KUKA KRL program: vw_prc_usr_r.src, vw_prc_usr_r.dat

--- vw_prc_usr_r.src ---
&ACCESS RV1
&COMMENT KS26
&REL 200
&PARAM DISKPATH = VW_User/Applikation/LM_Vision/Perceptron
&PARAM TPUSER_VERSION = 8.3.0
DEF vw_prc_usr_r( )
;
;*---------------------------------------------*
;* Perceptron GmbH                             *
;* Version 1.2.0  / VKRC 2 / VKRC 4            *
;*                                             *
;* Bearbeitet am:                              *
;* 21.12.2010 MG                               *
;*     ueberarbeitet auf Stand V1.0.0 / VKRC 4 *
;*                                             *
;* 26.12.2013 HF                               *
;*     512 Kompensations-UP holen neu          *
;*     521 Messpunkte abgeschlossen neu        *
;*     531 Messende mit SPS entfernt           *
;*     512 ist jetzt 514                       *
;*     FLAG-Modell-Kontrolle                   *
;*                                             *
;* 05.02.2014 MG                               *
;*     V1.1.6: VKRC4 mit                       *
;*             Robotertausch                   *
;*             Sensortausch                    *
;*             Compmodell                      *
;*     V1.1.7: Tempcompsystem                  *
;*                                             *
;* 15.07.2015 RB                               *
;*     V1.1.8: Modell-Erweiterung              *
;*             Modell-Flags angepasst          *
;*             UP-Nr.-Zuweiung angepasst       *
;*             Roboter Korrekturframe holen    *
;*                                             *
;* 12.12.2015 DB                               *
;*     Conveyor implementiert                  *
;*                                             *
;* 09.05.2017 HF                               *
;*     PRCP/Init implementiert                 *
;*                                             *
;*     V1.2.0: 524 - Achswinkel speichern      *
;*             525 - Start Messpunkt ID        *
;*                    Sendet Pose-ID           *
;*             SysInit-1  System Init          *
;*             SysInit-2  System Init          *
;*             ModelInit  Modellfreigaben      *
;*             FrameInit Max  VF-Limits        *
;*             FrameInit Min  VF-Limits        *
;*                                             *
;* 01.02.2019 HF                               *
;*     V1.3.0: TPUSER_VERSION = 8.3.0          *
;*                                             *
;*---------------------------------------------*
;
END
;
;FOLD Perceptron Interface
GLOBAL DEF PRC_Interface(USER_CMD:IN,CMD_SEL:IN,FUNKTION:IN,nPAR2:IN,nPAR3:IN,nPAR4:IN,nPAR5:IN,nPAR6:IN,nPAR7:IN,nPAR8:IN,nPAR9:IN)
DECL VW_USER_CMD USER_CMD
DECL INT         CMD_SEL      ; Modus
DECL INT         FUNKTION     ; Funktion
DECL INT         nPAR2
DECL INT         nPAR3
DECL INT         nPAR4
DECL INT         nPAR5
DECL INT         nPAR6
DECL INT         nPAR7
DECL INT         nPAR8
DECL INT         nPAR9
DECL INT         nFlagCounter
DECL INT         I ;allgemeiner Zaehler
DECL KRLMSG_T      USER_MSG
  IF USER_CMD == #USR_MAKRO THEN
     SWITCH CMD_SEL
        CASE 1001 ; PRC_SYSINIT_1      Hauptgruppe 9, Untergruppe 1
           ; System Einstellungen 1
           PRC_SysInit1(FUNKTION,nPAR2,nPAR3,nPAR4,nPAR5,nPAR6)
		     ; Subsystem              Toolkalibrier-Modus = 0-ToolFinder/1=Temperaturkalibrierung
	         ; Conveyortech           0=Ohne/1=Mit
             ; Alive-Bit              0=Ohne/1=Mit
             ; KorrekturBase          (Default 31, Conveyor 11)
		     ; Robotertausch-VF
           ; Frei
        CASE 1002 ; PRC_SYSINIT_2      Hauptgruppe 9, Untergruppe 2
           ; System Einstellungen 2
           PRC_SysInit2(FUNKTION,nPAR2,nPAR3,nPAR4,nPAR5,nPAR6)
		     ; Timeout Messpunkt      [ms]
		     ; Timeout Kommunikation  [ms]
		     ; Start Fehler-Flags
		     ; Start Master-Signale
		     ; Interrupt fuer RobMove
           ; Interrupt fuer RobNoMove
        CASE 1003 ; PRC_MODELINIT      Hauptgruppe 9, Untergruppe 3
           ; Modell Freigaben
           PRC_ModelInit(FUNKTION,nPAR2,nPAR3,nPAR4,nPAR5,nPAR6)
             ; Freigegebenes Modell
		     ; Freigegebenes Modell
		     ; Freigegebenes Modell
		     ; Freigegebenes Modell
		     ; Freigegebenes Modell
             ; Freigegebenes Modell
        CASE 1004 ; PRC_FRAMEINIT_MIN  Hauptgruppe 9, Untergruppe 4
           ; VF Limits
           PRC_FrameInit(0,0,FUNKTION,nPAR2,nPAR3,0)
           PRC_FrameInit(0,1,nPAR4,nPAR5,nPAR6,0)
             ; Min/Max                 0=Minimalgrenze / 1=Maximalgrenze
		     ; Trans/Rot               0=Translation   / 1=Rotation
		     ; X-Limit/A-Limit
		     ; Y-Limit/B-Limit
		     ; Z-Limit/C-Limit
             ; Frei
        CASE 1005 ; PRC_FRAMEINIT_MAX  Hauptgruppe 9, Untergruppe 5
           ; VF Limits
           PRC_FrameInit(1,0,FUNKTION,nPAR2,nPAR3,0)
           PRC_FrameInit(1,1,nPAR4,nPAR5,nPAR6,0)
             ; Min/Max                 0=Minimalgrenze / 1=Maximalgrenze
		     ; Trans/Rot               0=Translation   / 1=Rotation
		     ; X-Limit/A-Limit
		     ; Y-Limit/B-Limit
		     ; Z-Limit/C-Limit
             ; Frei
        DEFAULT
             ;
      ENDSWITCH ; CMD_SEL
      RETURN
  ENDIF
  IF USER_CMD <> #USR_INIT THEN
	SWITCH CMD_SEL
      CASE 1001 ; IMT  Hauptgruppe 9, Untergruppe 1
        N_PRC_Fkt = CMD_SEL
        SWITCH FUNKTION
          CASE 501,510,511,512,513,514,520,521,522,523,524,525,530,540,545,550,551,552,553,554,598,599
            ; OK
          DEFAULT
            N_PRC_MsgOff     = 900
            B_PRC_MsgFlg     = TRUE
            N_PRC_Err1       = 902   ; Funktion P1 ungueltig
            N_PRC_Ret1       = PRC_MsgErr(#NotifyMsg,N_PRC_Err1,FUNKTION,CMD_SEL)
            $FLAG[F_PRC_Err] = TRUE
            RETURN
        ENDSWITCH ; FUNKTION
      CASE 1002 ; RF  Hauptgruppe 9, Untergruppe 2
        N_PRC_Fkt = CMD_SEL
        SWITCH FUNKTION
          CASE 501,510,511,512,520,521,522,523,525,530,540,545,552,553,554,598,599
            ; OK
          DEFAULT
          N_PRC_MsgOff     = 900
          B_PRC_MsgFlg     = TRUE
          N_PRC_Err1       = 902 ; Funktion P1 ungueltig
          N_PRC_Ret1       = PRC_MsgErr(#NotifyMsg,N_PRC_Err1,FUNKTION,CMD_SEL)
          $FLAG[F_PRC_Err] = TRUE
          RETURN
        ENDSWITCH ; FUNKTION
      CASE 1003 ; AGauge  Hauptgruppe 9, Untergruppe 3
        N_PRC_Fkt = CMD_SEL
        SWITCH FUNKTION
          CASE 501,510,511,530,598,599
            ; OK
          DEFAULT
          N_PRC_MsgOff     = 900
          B_PRC_MsgFlg     = TRUE
          N_PRC_Err1       = 902   ; Funktion P1 ungueltig
          N_PRC_Ret1       = PRC_MsgErr(#NotifyMsg,N_PRC_Err1,FUNKTION,CMD_SEL)
          $FLAG[F_PRC_Err] = TRUE
          RETURN
        ENDSWITCH ; FUNKTION
      DEFAULT
        N_PRC_MsgOff     = 900
        B_PRC_MsgFlg     = TRUE
        N_PRC_Err1       = 1001   ; Modus P2 ungueltig
        N_PRC_Ret1       = PRC_MsgErr(#NotifyMsg,N_PRC_Err1,CMD_SEL,N_PRC_Ret1)
        $FLAG[F_PRC_Err] = TRUE
        RETURN
    ENDSWITCH ; CMD_SEL
  ENDIF ; USER_CMD
;
; ;FOLD USER_CMD
;
  SWITCH USER_CMD
    CASE #USR_INIT
      N_PRC_MsgOff = 50
      B_PRC_MsgFlg = FALSE
      B_PRC_RetVal = PRC_Sync()
;
;ENDFOLD (USER_CMD)
;
; ;FOLD Advance
;
  CASE #USR_ADV
	SWITCH N_PRC_Fkt
      CASE 1001 ; Hauptgruppe 9, Untergruppe 1
        ;PRC_IMTInterface
        N_PRC_Err1   = 0
        N_PRC_Err2   = 0
        N_PRC_UpNr   = 0
        N_PRC_MsgOff = 0
        B_PRC_MsgFlg = FALSE
        FOR nFlagCounter = N_PRC_FiErr TO N_PRC_FiErr + N_PRC_LgErr
          $FLAG[nFlagCounter] = FALSE
        ENDFOR
        N_PRC_Err1 = PRC_CheckParams(nPAR2,nPAR3,nPAR4,nPAR5,nPAR6,nPAR7,nPAR8)
        IF N_PRC_Err1 > 0 THEN
          N_PRC_Ret1 = PRC_MsgErr(#DlgMsg,N_PRC_Err1)
          $FLAG[F_PRC_Err] = TRUE
          RETURN
        ENDIF
        SWITCH FUNKTION
          CASE 553 ;korrektur ausfuehren
            USER_MSG.MSG_TXT[] = "553: ADV Step-1"
		    PRC_DebugDlg(8,0,0)
		    USER_MSG.MSG_TXT[] = "553: ADV Step-2"
            PRC_SetKorrektur(nPAR4)
		    USER_MSG.MSG_TXT[] = "553: ADV Step-3"
            N_PRC_Ret1 = PRC_MsgErr(#NotifyMsg,N_PRC_Err1)
		    USER_MSG.MSG_TXT[] = "553: ADV Step-4"
	      DEFAULT
			;
		ENDSWITCH ; FUNKTION
      CASE 1002 ; Hauptgruppe 9, Untergruppe 2
        PRC_AutoGuideInterface(#USR_ADV,CMD_SEL,FUNKTION,nPAR2,nPAR3,nPAR4,nPAR5,nPAR6,nPAR7,nPAR8,nPAR9)
      CASE 1003 ; Hauptgruppe 9, Untergruppe 3
        PRC_AutoGaugeInterface(#USR_ADV,CMD_SEL,FUNKTION,nPAR2,nPAR3,nPAR4,nPAR5,nPAR6,nPAR7,nPAR8,nPAR9)
    ENDSWITCH ; N_PRC_Fkt
;
;ENDFOLD (Advance)
;
  CASE #USR_TRIG
;
;FOLD Trig
;
    SWITCH N_PRC_Fkt
      CASE 1001 ; Hauptgruppe 9, Untergruppe 1
        ;PRC_IMTInterface
        SWITCH FUNKTION
          CASE 523 ; Scanning stoppen
            N_PRC_MsgOff = 250
            B_PRC_MsgFlg = FALSE
            REPEAT
              N_PRC_Err1 = PRC_EndScan(nPAR4)
              N_PRC_Ret1 = PRC_MsgErr(#NotifyMsg,N_PRC_Err1)
            UNTIL (N_PRC_Ret1 == 1)
            IF B_PRC_MsgFlg == TRUE THEN
              $FLAG[F_PRC_Err]   = TRUE
            ELSE
              $FLAG[F_PRC_NoErr] = TRUE
            ENDIF
          DEFAULT
		    ;
        ENDSWITCH ; FUNKTION
      CASE 1002 ; Hauptgruppe 9, Untergruppe 2
        PRC_AutoGuideInterface(#USR_TRIG,CMD_SEL,FUNKTION,nPAR2,nPAR3,nPAR4,nPAR5,nPAR6,nPAR7,nPAR8,nPAR9)
      CASE 1003 ; Hauptgruppe 9, Untergruppe 3
        PRC_AutoGaugeInterface(#USR_TRIG,CMD_SEL,FUNKTION,nPAR2,nPAR3,nPAR4,nPAR5,nPAR6,nPAR7,nPAR8,nPAR9)
    ENDSWITCH ; N_PRC_Fkt
;
;ENDFOLD (Trig)
;
  CASE #USR_MAIN
;
;FOLD Main
;
    SWITCH N_PRC_Fkt
      CASE 1001  ; Hauptgruppe 9, Untergruppe 1
        ; PRC_IMTInterface #USR_MAIN
        ;PRC_MainPrg
        N_PRC_PktNr  = nPAR4
	     N_PRC_BasNr  = $ACT_BASE
        N_PRC_TooNr  = $ACT_TOOL
        B_PRC_Ghost  = $IN[N_PRC_Ghost]
        ; bei Geisterschicht nur Messung starten, da
        ; dabei auch UP mit Punktmessung gestartet wird
        IF ((B_PRC_Ghost) AND (FUNKTION <> 510)) THEN
          $FLAG[F_PRC_Err]   = FALSE
          $FLAG[F_PRC_NoErr] = TRUE
          RETURN
        ENDIF
        SWITCH FUNKTION
          CASE 501 ; Statusanforderung
            N_PRC_MsgOff   = 300
            REPEAT
              N_PRC_Err1   = 1
              B_PRC_MsgFlg = FALSE
              N_PRC_Status = PRC_GetStatus()
              PRC_DebugDlg(1,N_PRC_Status,0)
              SWITCH N_PRC_Status
                CASE 300
                  ; OK
                CASE 301,306,307,308,309,317,318,323,324,327,328,329,330,343
                  B_PRC_MsgFlg = TRUE
                DEFAULT
                  N_PRC_Status = 309
                  B_PRC_MsgFlg = TRUE
              ENDSWITCH ; N_PRC_Status
              IF B_PRC_MsgFlg THEN
                N_PRC_Ret1 = PRC_MsgErr(#NotifyMsg,N_PRC_Status)
              ENDIF
              IF N_PRC_Status <> 300 THEN
                N_PRC_Ret1 = PRC_MsgErr(#NotifyMsg,345)
                IF N_PRC_Ret1 == 2 THEN
                  REPEAT
                    PRC_DebugDlg(9,0,0)
                    N_PRC_Err2 = PRC_Reset()
                    N_PRC_Ret2 = PRC_MsgErr(#NotifyMsg,N_PRC_Err2)
                  UNTIL (N_PRC_Ret2 == 1)
                ENDIF
              ELSE
                N_PRC_Ret1 = PRC_MsgErr(#NotifyMsg,1,N_PRC_Status)
              ENDIF
            UNTIL (N_PRC_Ret1 == 1)
            IF (B_PRC_MsgFlg == TRUE) THEN
              $FLAG[F_PRC_Err]   = TRUE
              $FLAG[F_PRC_NoErr] = FALSE
            ELSE
              $FLAG[F_PRC_Err]   = FALSE
              $FLAG[F_PRC_NoErr] = TRUE
            ENDIF
          CASE 510,514 ; Messung mit Punktmessung starten
            N_PRC_MsgOff = 100
            B_PRC_MsgFlg = FALSE
            IF (FUNKTION == 514) THEN
              O_PRC_CmpStr = TRUE
            ENDIF
            PRC_DebugDlg(6,0,0)
            PRC_DebugDlg(25,nPAR2,nPAR3)
            IF (PRC_StartMsrPktMsr(nPAR2,nPAR3,nPAR6) == N_PRC_MsgOff) THEN
              $FLAG[F_PRC_NoErr] = TRUE
            ELSE
              $FLAG[F_PRC_Err]   = TRUE
            ENDIF
            O_PRC_CmpStr = FALSE
          CASE 511 ; Mess UP-Nummer holen fuer Punktmessung
            N_PRC_MsgOff = 800
            B_PRC_MsgFlg = FALSE
            PRC_DebugDlg(24,0,0)
            N_PRC_Ret1 = PRC_GetMessUpNr(nPAR2,nPAR3,nPAR6)
            SWITCH N_PRC_Ret1
              CASE 800
                ; OK
              CASE 801,807,829,840,841
                $FLAG[F_PRC_Err] = TRUE
                B_PRC_MsgFlg     = TRUE
              DEFAULT
                $FLAG[F_PRC_Err] = TRUE
                B_PRC_MsgFlg     = TRUE
            ENDSWITCH ; N_PRC_Ret1
          CASE 512 ; Kompensations UP-Nummer holen fuer Punktmessung
            N_PRC_MsgOff = 800
            B_PRC_MsgFlg = FALSE
            PRC_DebugDlg(24,0,0)
            N_PRC_Ret1 = PRC_GetKompUpNr(nPAR2,nPAR3,nPAR6)
            SWITCH N_PRC_Ret1
              CASE 800,850,851,852,853,860,861
                ; OK
              CASE 801,807,809,811,829,840,841,843,870,871
                $FLAG[F_PRC_Err] = TRUE
                B_PRC_MsgFlg     = TRUE
              DEFAULT
                $FLAG[F_PRC_Err] = TRUE
                B_PRC_MsgFlg     = TRUE
            ENDSWITCH ; N_PRC_Ret1
          CASE 513 ; Messen komplett
            N_PRC_MsgOff = 100
            B_PRC_MsgFlg = FALSE
            N_PRC_Ret1 = PRC_MsgErr(#NotifyMsg,910,FUNKTION,CMD_SEL)
          CASE 520 ;Punktmessung starten
            N_PRC_MsgOff = 200
            B_PRC_MsgFlg = FALSE
            REPEAT
              PRC_DebugDlg(3,N_PRC_PktNr,0)
		      PRC_PunktMessung(N_PRC_PktNr,-1,-1)
              N_PRC_Ret1 = PRC_MsgErr(#NotifyMsg,N_PRC_Err1,0,N_PRC_PktNr)
            UNTIL (N_PRC_Ret1 == 1)
            IF B_PRC_MsgFlg THEN
              $FLAG[F_PRC_Err]   = TRUE
            ELSE
              $FLAG[F_PRC_NoErr] = TRUE
            ENDIF
          CASE 521 ; Punkte beendet
            N_PRC_MsgOff = 200
            B_PRC_MsgFlg = FALSE
            REPEAT
              PRC_DebugDlg(3,N_PRC_LstPkt,0)
              PRC_PunktMessung(N_PRC_LstPkt,-1,-1)
              N_PRC_Ret1 = PRC_MsgErr(#NotifyMsg,N_PRC_Err1,0,N_PRC_LstPkt)
            UNTIL (N_PRC_Ret1 == 1)
            IF B_PRC_MsgFlg THEN
              $FLAG[F_PRC_Err]   = TRUE
            ELSE
              $FLAG[F_PRC_NoErr] = TRUE
            ENDIF
          CASE 522 ;Scanning starten
            N_PRC_MsgOff = 250
            B_PRC_MsgFlg = FALSE
            REPEAT
              N_PRC_Err1 = 0
              PRC_StartScan(N_PRC_PktNr)
              N_PRC_Ret1 = 1
              N_PRC_Ret1 = PRC_MsgErr(#NotifyMsg,N_PRC_Err1)
            UNTIL (N_PRC_Ret1 == 1)
            IF B_PRC_MsgFlg THEN
              $FLAG[F_PRC_Err]   = TRUE
            ELSE
              $FLAG[F_PRC_NoErr] = TRUE
            ENDIF
          CASE 523
            ; in TRIG ausgelagert
          CASE 524 ;Achswinkel speichern
            wait for TRUE
            IF ((N_PRC_PktNr > 0) and (N_PRC_PktNr <=100)) THEN
              AX_PRC_Pose[N_PRC_PktNr]=$Axis_act
            ENDIF
          CASE 525 ;Sende Pose-ID
		      N_PRC_MsgOff = 200
            B_PRC_MsgFlg = FALSE
            REPEAT
              PRC_DebugDlg(3,N_PRC_PktNr,0)
		        PRC_PunktMessung(N_PRC_PktNr,N_PRC_BasNr,N_PRC_TooNr)
              N_PRC_Ret1 = PRC_MsgErr(#NotifyMsg,N_PRC_Err1,0,N_PRC_PktNr)
            UNTIL (N_PRC_Ret1 == 1)
            IF B_PRC_MsgFlg THEN
              $FLAG[F_PRC_Err]   = TRUE
            ELSE
              $FLAG[F_PRC_NoErr] = TRUE
            ENDIF
          CASE 530 ;Messung beenden
            N_PRC_MsgOff = 400
            B_PRC_MsgFlg = FALSE
            N_PRC_Err1   =  1
            PRC_DebugDlg(4,0,0)
            PRC_MessungBeenden(CMD_SEL)
            N_PRC_Ret1 = PRC_MsgErr(#NotifyMsg,N_PRC_Err1)
            IF B_PRC_MsgFlg THEN
              $FLAG[F_PRC_Err]   = TRUE
            ELSE
              $FLAG[F_PRC_NoErr] = TRUE
            ENDIF
          CASE 540 ;Sensortausch (Messung mit Punktmessung)
            PRC_DebugDlg(5,0,0)
            N_PRC_MsgOff = 600
            B_PRC_MsgFlg = FALSE
            B_PRC_1Kalib = FALSE
            B_PRC_TmpKalib = FALSE
            B_PRC_ToFiOK=FALSE
            IF (($mode_op <> #T1) AND ($mode_op <> #T2)) THEN
              N_PRC_Err1   = 639
              B_PRC_MsgFlg = TRUE
              N_PRC_Ret1   = PRC_MsgErr(#NotifyMsg,N_PRC_Err1)
              $FLAG[F_PRC_Err] = TRUE
              RETURN
            ENDIF
            LOOP
              REPEAT ; Sensorpruefung
                N_PRC_ModNr = N_PRC_SenPrM
                N_PRC_UpNr  = N_PRC_SenPrU
                REPEAT
                  N_PRC_Err1   = 0
                  N_PRC_Ret1   = 1
                  B_PRC_MsgFlg = FALSE
                  N_PRC_Status = PRC_GetStatus()
                  PRC_DebugDlg(1,N_PRC_Status,0)
                  IF B_PRC_MsgFlg THEN
                    N_PRC_Ret1 = PRC_MsgErr(#NotifyMsg,N_PRC_Status)
                    RETURN
                  ELSE
                    IF (N_PRC_Status <> 600) THEN
                      N_PRC_Status=606
                      N_PRC_Ret1   = PRC_MsgErr(#NotifyMsg,N_PRC_Status)
                      SWITCH N_PRC_Ret1
                        CASE 1
                          N_PRC_Ret1   = PRC_MsgErr(#NotifyMsg,644)
                          return
                        CASE 2
                          N_PRC_Ret1   = 0
                        DEFAULT
                          ;falsche Dialogantwort
                          $FLAG[F_PRC_Err]   = TRUE
                          RETURN
                      ENDSWITCH ; N_PRC_Ret1
                    ELSE
                      N_PRC_Ret1 = 1
                    ENDIF
                  ENDIF
                UNTIL (N_PRC_Ret1 == 1)
                IF B_PRC_MsgFlg THEN
                  $FLAG[F_PRC_Err] = TRUE
                  RETURN
                ENDIF
                B_PRC_ISTOOL = TRUE
                PRC_DebugDlg(16,0,0)
                PRC_DebugDlg(25,N_PRC_ModNr,N_PRC_UpNr)
                N_PRC_MsrErg = PRC_StartMsrPktMsr(N_PRC_ModNr,N_PRC_UpNr,nPAR6)
                N_PRC_MsgOff = 600
                IF B_PRC_MsgFlg THEN
                  B_PRC_ISTOOL = FALSE
                  $FLAG[F_PRC_Err] = TRUE
                  RETURN
                ENDIF
                SWITCH N_PRC_MsrErg
            CASE 600,601  ;alles ok
              N_PRC_Ret1 = PRC_MsgErr(#NotifyMsg,633)
              B_PRC_ISTOOL = FALSE
              if B_PRC_1Kalib then ;min 1mal kalib
                B_PRC_ToFiOK=TRUE
                if ((N_PRC_SubSystem == 1) and not B_PRC_TmpKalib) then
                  ;Tempkalib ausfuehren
                else
                  N_PRC_Ret1 = PRC_MsgErr(#NotifyMsg,698)
                  $FLAG[F_PRC_NoErr] = TRUE
                  RETURN
                endif
              endif
            CASE 1151, 1152, 1155, 1156   ; Kalibrierung erforderlich
              N_PRC_RET1 = 1
            CASE 603, 605, 606, 607, 1153, 1154, 1157, 1158   ; Sensormontage pruefen
              N_PRC_MsrErg = 610
              N_PRC_Ret1   = PRC_MsgErr(#NotifyMsg,N_PRC_MsrErg)
              IF N_PRC_Ret1 == 1 THEN
                B_PRC_ISTOOL = FALSE
                $FLAG[F_PRC_Err] = TRUE
                RETURN
              ENDIF
            DEFAULT
              N_PRC_Ret1 = PRC_MsgErr(#NotifyMsg,N_PRC_Err1)
              B_PRC_ISTOOL = FALSE
              $FLAG[F_PRC_Err] = TRUE
              RETURN
            ENDSWITCH
          UNTIL N_PRC_Ret1 == 1
          B_PRC_ISTOOL = FALSE
          if (((N_PRC_SubSystem == 1) and (B_PRC_ToFiOK)) OR (N_PRC_SubSystem == 0))then
            N_PRC_Ret1   = PRC_MsgErr(#NotifyMsg,630)
          else
            N_PRC_Ret1   = PRC_MsgErr(#NotifyMsg,650)
          endif
          REPEAT
            N_PRC_Err1   = 0
            B_PRC_MsgFlg = FALSE
            N_PRC_Status = PRC_GetStatus()
            PRC_DebugDlg(1,N_PRC_Status,0)
            IF ((N_PRC_SubSystem == 1) AND NOT(B_PRC_ToFiOK)) THEN
              if (N_PRC_Status <> 630) then
                N_PRC_Err1   = 652   ; Perceptron nicht in Toolfinder-Modus
                B_PRC_MsgFlg = TRUE
              endif
            endif
            IF ((N_PRC_SubSystem <> 1) OR ((N_PRC_SubSystem == 1) AND (B_PRC_ToFiOK))) then
              if(N_PRC_Status <> 623) THEN
                N_PRC_Err1   = 632   ; Perceptron nicht in Kalibrier-Modus
                B_PRC_MsgFlg = TRUE
              endif
            endif
            IF B_PRC_MsgFlg THEN
              N_PRC_Ret1 = PRC_MsgErr(#NotifyMsg,N_PRC_Err1)
            ELSE
              N_PRC_Ret1   = 1
            ENDIF
          UNTIL (N_PRC_Ret1 == 1)
          IF (B_PRC_MsgFlg) THEN
            $FLAG[F_PRC_Err] = TRUE
            RETURN
          ENDIF
          IF (((N_PRC_SubSystem == 1) and B_PRC_ToFiOK) OR (N_PRC_SubSystem == 0)) then
            N_PRC_ModNr = N_PRC_TmpCmpM
            N_PRC_UpNr  = N_PRC_TmpCmpU
            B_PRC_TmpKalib = TRUE
          else
            N_PRC_ModNr = N_PRC_SenTaM
            N_PRC_UpNr  = N_PRC_SenTaU
          endif
          PRC_DebugDlg(26,0,0)
          PRC_DebugDlg(25,N_PRC_ModNr,N_PRC_UpNr)
          N_PRC_MsrErg = PRC_StartMsrPktMsr(N_PRC_ModNr,N_PRC_UpNr,nPAR6) ; Starten im Toolfinder od. Kalib-Modus
          N_PRC_MsgOff = 600
          IF B_PRC_MsgFlg THEN
            N_PRC_Ret1       = PRC_MsgErr(#NotifyMsg,N_PRC_Err1)
            $FLAG[F_PRC_Err] = TRUE
            RETURN
          ENDIF
          IF (((N_PRC_SubSystem == 1) and B_PRC_ToFiOK)  OR (N_PRC_SubSystem == 0)) then
            N_PRC_Ret1 = PRC_MsgErr(#NotifyMsg,699)
          ELSE
            N_PRC_Ret1 = PRC_MsgErr(#NotifyMsg,653)
          ENDIF
          B_PRC_1Kalib = TRUE
        ENDLOOP
      CASE 545 ;Robotertausch
        PRC_DebugDlg(10,0,0)
        N_PRC_MsgOff   = 700
        B_PRC_MsgFlg   = FALSE
        B_PRC_TmpKalib = FALSE
        B_PRC_ToFiOK   = FALSE
        B_PRC_NoBaKo   = FALSE
        IF (($mode_op <> #T1) AND ($mode_op <> #T2)) THEN
          N_PRC_Err1 = 739
          B_PRC_MsgFlg = TRUE
          N_PRC_Ret1 = PRC_MsgErr(#NotifyMsg,N_PRC_Err1)
          $FLAG[F_PRC_Err] = TRUE
          RETURN
        ENDIF
        REPEAT ; Roboterpruefung
          N_PRC_ModNr = N_PRC_RobPrM
          N_PRC_UpNr  = N_PRC_RobPrU
          REPEAT
            N_PRC_Err1   = 0
            N_PRC_Ret1   = 1
            B_PRC_MsgFlg = FALSE

            N_PRC_Status = PRC_GetStatus()
            PRC_DebugDlg(1,N_PRC_Status,0)
            IF B_PRC_MsgFlg THEN
              N_PRC_Ret1 = PRC_MsgErr(#NotifyMsg,N_PRC_Status)
              RETURN
            ELSE
              IF (N_PRC_Status <> 700) THEN
                N_PRC_Ret1   = PRC_MsgErr(#NotifyMsg,N_PRC_Status)
                SWITCH N_PRC_Ret1
                CASE 1
                  N_PRC_Ret1   = PRC_MsgErr(#NotifyMsg,744)
                  RETURN
                CASE 2
                  N_PRC_Ret1   = 0
                DEFAULT
                  ;falsche Dialogantwort
                  $FLAG[F_PRC_Err]   = TRUE
                  RETURN
                ENDSWITCH
              ELSE
                N_PRC_Ret1 = 1
              ENDIF
            ENDIF
          UNTIL(N_PRC_Ret1 == 1)
          IF B_PRC_MsgFlg THEN
            $FLAG[F_PRC_Err] = TRUE
            RETURN
          ENDIF
          B_PRC_ISBASE = TRUE
          PRC_DebugDlg(6,0,0)
          PRC_DebugDlg(25,N_PRC_ModNr,N_PRC_UpNr)
          N_PRC_MsrErg = PRC_StartMsrPktMsr(N_PRC_ModNr,N_PRC_UpNr,nPAR6)
          N_PRC_MsgOff = 700
          IF B_PRC_MsgFlg THEN
            B_PRC_ISBASE = FALSE
            $FLAG[F_PRC_Err] = TRUE
            RETURN
          ENDIF
          SWITCH N_PRC_MsrErg
          CASE 700, 1152, 1156; alles ok. ,Sensortoleranz
            if (N_PRC_MsrErg == 700) then
              ;N_PRC_Ret1 = PRC_MsgErr(#NotifyMsg,733)
            endif
            B_PRC_ISBASE = FALSE
            ;---------Sensortausch -----------------------------
            PRC_DebugDlg(5,0,0)
            N_PRC_MsgOff = 600
            B_PRC_MsgFlg = FALSE
            B_SensIsKalib = FALSE
            IF (($mode_op <> #T1) AND ($mode_op <> #T2)) THEN
              N_PRC_Err1   = 639
              B_PRC_MsgFlg = TRUE
              N_PRC_Ret1   = PRC_MsgErr(#NotifyMsg,N_PRC_Err1)
              $FLAG[F_PRC_Err] = TRUE
              RETURN
            ENDIF
            Repeat
              ;-------------Sensorkalibrierung-------------------
              B_PRC_ISTOOL = FALSE
              IF (N_PRC_SubSystem==1) THEN
                N_PRC_Ret1   = PRC_MsgErr(#NotifyMsg,650)
              ELSE
                N_PRC_Ret1   = PRC_MsgErr(#NotifyMsg,630)
              ENDIF
              REPEAT
                N_PRC_Err1   = 0
                B_PRC_MsgFlg = FALSE
                N_PRC_Status = PRC_GetStatus()
                PRC_DebugDlg(1,N_PRC_Status,0)
                IF (N_PRC_SubSystem == 1) THEN
                  if (N_PRC_Status <> 630) then
                    N_PRC_Err1   = 652   ; Perceptron nicht in Toolfinder-Modus
                    B_PRC_MsgFlg = TRUE
                  endif
                endif
                IF (N_PRC_SubSystem <> 1) then
                  if(N_PRC_Status <> 623) THEN
                    N_PRC_Err1   = 632   ; Perceptron nicht in Kalibrier-Modus
                    B_PRC_MsgFlg = TRUE
                  endif
                endif
                IF B_PRC_MsgFlg THEN
                  N_PRC_Ret1 = PRC_MsgErr(#NotifyMsg,N_PRC_Err1)
                ELSE
                  N_PRC_Ret1   = 1
                ENDIF
              UNTIL (N_PRC_Ret1 == 1)
              IF (B_PRC_MsgFlg) THEN
                $FLAG[F_PRC_Err] = TRUE
                RETURN
              ENDIF
              IF (N_PRC_SubSystem == 1) then
                N_PRC_ModNr = N_PRC_SenTaM
                N_PRC_UpNr  = N_PRC_SenTaU
              else
                N_PRC_ModNr = N_PRC_TmpCmpM
                N_PRC_UpNr  = N_PRC_TmpCmpU
              endif
              PRC_DebugDlg(26,0,0)
              PRC_DebugDlg(25,N_PRC_ModNr,N_PRC_UpNr)
              N_PRC_MsrErg = PRC_StartMsrPktMsr(N_PRC_ModNr,N_PRC_UpNr,nPAR6) ; Starten im Toolfinder-Modus
              N_PRC_MsgOff = 600
              IF B_PRC_MsgFlg THEN
                N_PRC_Ret1       = PRC_MsgErr(#NotifyMsg,N_PRC_Err1)
                $FLAG[F_PRC_Err] = TRUE
                RETURN
              ENDIF
              SWITCH N_PRC_MsrErg
              CASE 600,601  ;alles ok
                ;N_PRC_Ret1 = PRC_MsgErr(#NotifyMsg,699)
                $FLAG[F_PRC_NoErr] = TRUE
                B_SensIsKalib = TRUE
              CASE 1151, 1152, 1155, 1156   ; Kalibrierung erforderlich
                N_PRC_RET1 = 1
              CASE 603, 605, 606, 607, 1153, 1154, 1157, 1158   ; Sensormontage pruefen
                N_PRC_MsrErg = 610
                N_PRC_Ret1   = PRC_MsgErr(#NotifyMsg,N_PRC_MsrErg)
                IF N_PRC_Ret1 == 1 THEN
                  B_PRC_ISTOOL = FALSE
                  $FLAG[F_PRC_Err] = TRUE
                  RETURN
                ENDIF
              DEFAULT
                N_PRC_Ret1 = PRC_MsgErr(#NotifyMsg,N_PRC_Err1)
                B_PRC_ISTOOL = FALSE
                $FLAG[F_PRC_Err] = TRUE
                RETURN
              ENDSWITCH
              Until B_SensIsKalib
            IF (N_PRC_SubSystem == 1) then
              N_PRC_Ret1 = PRC_MsgErr(#NotifyMsg,796)
            else
              ;                 N_PRC_Ret1 = PRC_MsgErr(#NotifyMsg,699)
            ENDIF
            ;---------------ende Sensorkalibrierung-------------------
            N_PRC_MsgOff = 700
            B_PRC_MsgFlg = FALSE
          CASE 703, 705, 706, 707, 1151, 1152, 1153, 1154, 1155, 1157, 1158   ;Robotermontage pruefen
            N_PRC_MsrErg = 710
            N_PRC_Ret1 = PRC_MsgErr(#NotifyMsg,N_PRC_MsrErg)
            IF N_PRC_Ret1 == 1 THEN
              B_PRC_ISBASE = FALSE
              $FLAG[F_PRC_Err] = TRUE
              RETURN
            ENDIF
          DEFAULT
            B_PRC_ISBASE = FALSE
            N_PRC_Ret1 = PRC_MsgErr(#NotifyMsg,N_PRC_Err1)
            $FLAG[F_PRC_Err] = TRUE
            RETURN
          ENDSWITCH
        UNTIL (N_PRC_Ret1 == 1)
        B_PRC_ISBASE = FALSE
        REPEAT
          REPEAT
            N_PRC_MsgOff = 700
            N_PRC_Err1   = PRC_MsgErr(#NotifyMsg,730)
            N_PRC_Err1   = 0
            B_PRC_MsgFlg = FALSE
            N_PRC_Status = PRC_GetStatus()
            PRC_DebugDlg(1,N_PRC_Status,0)
            IF (N_PRC_Status <> 700) THEN
              N_PRC_Err1   = 732 ; Perceptron nicht in Automtikmodus
              B_PRC_MsgFlg = TRUE
            ELSE
              B_PRC_MsgFlg = FALSE
              N_PRC_Ret1   = 1
            ENDIF
            IF B_PRC_MsgFlg THEN
              N_PRC_Ret1 = PRC_MsgErr(#NotifyMsg,N_PRC_Err1)
            ENDIF
          UNTIL (N_PRC_Ret1 == 1)
          IF (B_PRC_MsgFlg) THEN
            $FLAG[F_PRC_Err] = TRUE
            RETURN
          ENDIF
          N_PRC_ModNr  = N_PRC_RobTaM
          N_PRC_UpNr   = N_PRC_RobTaU
          PRC_DebugDlg(6,0,0)
          PRC_DebugDlg(25,N_PRC_ModNr,N_PRC_UpNr)
          N_PRC_MsrErg = PRC_StartMsrPktMsr(N_PRC_ModNr,N_PRC_UpNr,nPAR6)
          N_PRC_MsgOff = 700
          IF B_PRC_MsgFlg THEN
            N_PRC_Ret1 = PRC_MsgErr(#NotifyMsg,N_PRC_Err1)
            $FLAG[F_PRC_Err] = TRUE
            RETURN
          ENDIF
          SWITCH N_PRC_MsrErg
          CASE 700,701  ;alles ok
          ;N_PRC_Ret1 = PRC_MsgErr(#NotifyMsg,733)
          IF ((N_PRC_Subsystem == 1) and NOT(B_PRC_TMPKALIB)) THEN
            ;-------------Sensorkalibrierung-------------------
            B_SensIsKalib = FALSE
            N_PRC_MsgOff = 600
            N_PRC_Ret1   = PRC_MsgErr(#NotifyMsg,795)
            Repeat
              B_PRC_ISTOOL = FALSE
              N_PRC_Ret1   = PRC_MsgErr(#NotifyMsg,630)
              REPEAT
                N_PRC_Err1   = 0
                B_PRC_MsgFlg = FALSE
                N_PRC_Status = PRC_GetStatus()
                PRC_DebugDlg(1,N_PRC_Status,0)
                IF (N_PRC_Status <> 623) THEN ;kalibmode
                  N_PRC_Err1   = 632   ; Perceptron nicht in Kalibrier-Modus
                  B_PRC_MsgFlg = TRUE
                ELSE
                  B_PRC_MsgFlg = FALSE
                  N_PRC_Ret1   = 1
                ENDIF
                IF B_PRC_MsgFlg THEN
                  N_PRC_Ret1 = PRC_MsgErr(#NotifyMsg,N_PRC_Err1)
                ENDIF
              UNTIL (N_PRC_Ret1 == 1)
              IF (B_PRC_MsgFlg) THEN
                $FLAG[F_PRC_Err] = TRUE
                RETURN
              ENDIF
              N_PRC_ModNr = N_PRC_TmpCmpM
              N_PRC_UpNr  = N_PRC_TmpCmpU
              PRC_DebugDlg(26,0,0)
              PRC_DebugDlg(25,N_PRC_ModNr,N_PRC_UpNr)
              N_PRC_MsrErg = PRC_StartMsrPktMsr(N_PRC_ModNr,N_PRC_UpNr,nPAR6) ; Starten im Kalibrier-Modus
              N_PRC_MsgOff = 600
              IF B_PRC_MsgFlg THEN
                N_PRC_Ret1       = PRC_MsgErr(#NotifyMsg,N_PRC_Err1)
                $FLAG[F_PRC_Err] = TRUE
                RETURN
              ENDIF
              SWITCH N_PRC_MsrErg
              CASE 600,601  ;alles ok
                ;N_PRC_Ret1 = PRC_MsgErr(#NotifyMsg,699)
                $FLAG[F_PRC_NoErr] = TRUE
                B_SensIsKalib = TRUE
                B_PRC_TmpKalib = TRUE
              CASE 1152, 1156   ; Kalibrierung erforderlich
                N_PRC_RET1 = 1
              CASE 1153, 1154, 1157, 1158   ; Sensormontage pruefen
                N_PRC_MsrErg = 610
                N_PRC_Ret1   = PRC_MsgErr(#NotifyMsg,N_PRC_MsrErg)
                IF N_PRC_Ret1 == 1 THEN
                B_PRC_ISTOOL = FALSE
                $FLAG[F_PRC_Err] = TRUE
                RETURN
                ENDIF
              DEFAULT
                N_PRC_Ret1 = PRC_MsgErr(#NotifyMsg,N_PRC_Err1)
                B_PRC_ISTOOL = FALSE
                $FLAG[F_PRC_Err] = TRUE
                RETURN
              ENDSWITCH
            Until B_SensIsKalib
            ;---------------ende Sensorkalibrierung-------------------
          ENDIF
          B_PRC_ISBase = FALSE
          IF not(B_PRC_NoBaKo) then
            N_PRC_RET1   = 0
            B_PRC_NoBaKo = TRUE
          else
            N_PRC_RET1 = 1
          endif
          CASE 1151, 1152, 1155, 1156   ; Korrektur holen+aufrechnen
          N_PRC_Ret1 = PRC_MsgErr(#NotifyMsg,797)
          VF_PRC_RobKor = $BASE:AVF_PRC_Korr[N_PRC_VFNr]:INV_POS($BASE)
          ;halt ; VF_PRC_RobKor checken
          FOR I = 1 TO MAX_BASE
            BASE_DATA[I] = VF_PRC_RobKor:BASE_DATA[I]
          ENDFOR
          ;zum testen nur Base4
          ;BASE_DATA[4] = VF_PRC_RobKor:BASE_DATA[4]
          ;-------------Sensorkalibrierung-------------------
          N_PRC_MsgOff = 600
          N_PRC_Ret1   = PRC_MsgErr(#NotifyMsg,795)
          Repeat
            B_PRC_ISTOOL = FALSE
            N_PRC_Ret1   = PRC_MsgErr(#NotifyMsg,630)
            REPEAT
              N_PRC_Err1   = 0
              B_PRC_MsgFlg = FALSE
              N_PRC_Status = PRC_GetStatus()
              PRC_DebugDlg(1,N_PRC_Status,0)
              IF (N_PRC_Status <> 623) THEN ;kalibmode
                N_PRC_Err1   = 632   ; Perceptron nicht in Kalibrier-Modus
                B_PRC_MsgFlg = TRUE
              ELSE
                B_PRC_MsgFlg = FALSE
                N_PRC_Ret1   = 1
              ENDIF
              IF B_PRC_MsgFlg THEN
                N_PRC_Ret1 = PRC_MsgErr(#NotifyMsg,N_PRC_Err1)
              ENDIF
            UNTIL (N_PRC_Ret1 == 1)
            IF (B_PRC_MsgFlg) THEN
              $FLAG[F_PRC_Err] = TRUE
              RETURN
            ENDIF
            N_PRC_ModNr = N_PRC_TmpCmpM
            N_PRC_UpNr  = N_PRC_TmpCmpU
            PRC_DebugDlg(26,0,0)
            PRC_DebugDlg(25,N_PRC_ModNr,N_PRC_UpNr)
            N_PRC_MsrErg = PRC_StartMsrPktMsr(N_PRC_ModNr,N_PRC_UpNr,nPAR6)
            N_PRC_MsgOff = 600
            IF B_PRC_MsgFlg THEN
              N_PRC_Ret1       = PRC_MsgErr(#NotifyMsg,N_PRC_Err1)
              $FLAG[F_PRC_Err] = TRUE
              RETURN
            ENDIF
            SWITCH N_PRC_MsrErg
            CASE 600,601  ;alles ok
              ;N_PRC_Ret1 = PRC_MsgErr(#NotifyMsg,699)
              $FLAG[F_PRC_NoErr] = TRUE
              B_SensIsKalib = TRUE
              B_PRC_TmpKalib = TRUE
              N_PRC_RET1 = 2 ;damit wird nochmal pruefprogramm gefahren.
            CASE 1152, 1156   ; Kalibrierung erforderlich
              N_PRC_RET1 = 1
            CASE 1153, 1154, 1157, 1158   ; Sensormontage pruefen
              N_PRC_MsrErg = 610
              N_PRC_Ret1   = PRC_MsgErr(#NotifyMsg,N_PRC_MsrErg)
              IF N_PRC_Ret1 == 1 THEN
                B_PRC_ISTOOL = FALSE
                $FLAG[F_PRC_Err] = TRUE
                RETURN
              ENDIF
            DEFAULT
              N_PRC_Ret1 = PRC_MsgErr(#NotifyMsg,N_PRC_Err1)
              B_PRC_ISTOOL = FALSE
              $FLAG[F_PRC_Err] = TRUE
              RETURN
            ENDSWITCH
          Until B_SensIsKalib
          ;---------------ende Sensorkalibrierung-------------------
          N_PRC_MsgOff = 700
          N_PRC_RET1 = 0
          CASE 1151, 1154, 1155, 1158, 2000 ;Robotermontage pruefen
            N_PRC_MsrErg = 710
            N_PRC_Ret1 = PRC_MsgErr(#NotifyMsg,710)
            IF N_PRC_Ret1 == 1 THEN
              B_PRC_ISBASE = FALSE
              $FLAG[F_PRC_Err] = TRUE
              RETURN
            ENDIF
          DEFAULT
            N_PRC_Ret1 = PRC_MsgErr(#NotifyMsg,N_PRC_Err1)
            B_PRC_ISBase = FALSE
            $FLAG[F_PRC_Err] = TRUE
            RETURN
          ENDSWITCH
        UNTIL (N_PRC_RET1 == 1)

        N_PRC_Ret1 = PRC_MsgErr(#NotifyMsg,798)
        $FLAG[F_PRC_NoErr] = TRUE
      CASE 551 ;Messen, Korrketurwerte abholen, Korrektur ausfuehren
        N_PRC_MsgOff = 1000
        B_PRC_MsgFlg = FALSE
        N_PRC_Ret1 = PRC_MsgErr(#NotifyMsg,910,FUNKTION,CMD_SEL)
      CASE 552 ;Korrketurwerte abholen
        USER_MSG.MSG_TXT[] = "552: Main Step-1"
		N_PRC_MsgOff = 1000
        B_PRC_MsgFlg = FALSE
        PRC_DebugDlg(7,0,0)
        PRC_GetKorrektur(nPAR2,nPAR3,nPAR4,nPAR6)
		USER_MSG.MSG_TXT[] = "552: Main Step-2"
        SWITCH N_PRC_Ret1
        CASE 1000
          ; OK
        CASE 1001,1017,1018,1027,1028,1038,1042,1043
          B_PRC_MsgFlg = TRUE
        DEFAULT
          B_PRC_MsgFlg = TRUE
        ENDSWITCH
        N_PRC_Ret1 = PRC_MsgErr(#NotifyMsg,N_PRC_Err1)
		USER_MSG.MSG_TXT[] = "552: Main Step-3"
      CASE 553 ;Korrketur ausfuehren
        USER_MSG.MSG_TXT[] = "553: Main Step-1"
		N_PRC_MsgOff = 1000
        B_PRC_MsgFlg = FALSE
          ;wird im Advance erledigt, ins main geschoben HF
        PRC_DebugDlg(8,0,0)
        PRC_SetKorrektur(nPAR4)
        N_PRC_Ret1 = PRC_MsgErr(#NotifyMsg,N_PRC_Err1)
		USER_MSG.MSG_TXT[] = "553: Main Step-2"
      CASE 554   ;korrektur holen + ausfuehren
        N_PRC_MsgOff = 1000
        B_PRC_MsgFlg = FALSE
        PRC_DebugDlg(7,0,0)
        PRC_GetKorrektur(nPAR2,nPAR3,nPAR4,nPAR6)
        SWITCH N_PRC_Ret1
        CASE 1000
          ; OK
        CASE 1001,1017,1018,1027,1028,1038,1042,1043
          B_PRC_MsgFlg = TRUE
        DEFAULT
          B_PRC_MsgFlg = TRUE
        ENDSWITCH
        N_PRC_Ret1 = PRC_MsgErr(#NotifyMsg,N_PRC_Err1)
        N_PRC_MsgOff = 1000
        B_PRC_MsgFlg = FALSE
        PRC_DebugDlg(8,0,0)
        PRC_SetKorrektur(nPAR4)
        N_PRC_Ret1 = PRC_MsgErr(#NotifyMsg,N_PRC_Err1)
      CASE 598 ;Perceptron reset
        N_PRC_MsgOff = 500
        B_PRC_MsgFlg = FALSE
        PRC_DebugDlg(9,0,0)
        N_PRC_Err1   = PRC_Reset()
        N_PRC_Ret1   = 1
        N_PRC_Ret1   = PRC_MsgErr(#NotifyMsg,N_PRC_Err1)
        IF N_PRC_Err1 > 0 THEN
          $FLAG[F_PRC_Err]   = TRUE
        ELSE
          $FLAG[F_PRC_NoErr] = TRUE
        ENDIF
      CASE 599 ;Version
        B_PRC_MsgKri = TRUE
        N_PRC_Ret1   = PRC_MsgErr(#NotifyMsg,9000)
      ENDSWITCH
      ;ENDFOLD (Main IMT)
    CASE 1002  ; Hauptgruppe 9, Untergruppe 2
      PRC_AutoGuideInterface(#USR_MAIN,CMD_SEL,FUNKTION,nPAR2,nPAR3,nPAR4,nPAR5,nPAR6,nPAR7,nPAR8,nPAR9)
    CASE 1003  ; Hauptgruppe 9, Untergruppe 3
      PRC_AutoGaugeInterface(#USR_MAIN,CMD_SEL,FUNKTION,nPAR2,nPAR3,nPAR4,nPAR5,nPAR6,nPAR7,nPAR8,nPAR9)
    ENDSWITCH
    ;
    ;ENDFOLD (Main
    ;
  DEFAULT
    N_PRC_MsgOff = 900
    B_PRC_MsgFlg = TRUE
    N_PRC_Err1   = 911   ; Kommando ungueltig
    N_PRC_Ret1   = PRC_MsgErr(#NotifyMsg,N_PRC_Err1,CMD_SEL,N_PRC_Ret1)
    $FLAG[F_PRC_Err] = TRUE
    RETURN
  ENDSWITCH
END
;
  ;FOLD Roboter Fuehrung
;
GLOBAL DEF PRC_AutoGuideInterface(USER_CMD:IN,CMD_SEL:IN,FUNKTION:IN,nPAR2:IN,nPAR3:IN,nPAR4:IN,nPAR5:IN,nPAR6:IN,nPAR7:IN,nPAR8:IN,nPAR9:IN)
DECL VW_USER_CMD USER_CMD
DECL INT         CMD_SEL
DECL INT         FUNKTION
DECL INT         nPAR2
DECL INT         nPAR3
DECL INT         nPAR4
DECL INT         nPAR5
DECL INT         nPAR6
DECL INT         nPAR7
DECL INT         nPAR8
DECL INT         nPAR9
DECL INT         nFlagCounter
  SWITCH USER_CMD
    CASE #USR_ADV
;
    ;FOLD Advance
;
      N_PRC_UpNr = 0
      FOR nFlagCounter = N_PRC_FiErr TO N_PRC_FiErr + N_PRC_LgErr
        $FLAG[nFlagCounter] = FALSE
      ENDFOR
      N_PRC_Err1 = PRC_CheckParams(nPAR2,nPAR3,nPAR4,nPAR5,nPAR6,nPAR7,nPAR8)
      IF N_PRC_Err1 > 0 THEN
        N_PRC_Ret1 = PRC_MsgErr(#DlgMsg,N_PRC_Err1)
        $FLAG[F_PRC_Err]   = TRUE
        RETURN
      ENDIF
      SWITCH FUNKTION
        CASE 553   ;korrektur ausfuehren
          PRC_DebugDlg(8,0,0)
          PRC_SetKorrektur(nPAR4)
          N_PRC_Ret1 = PRC_MsgErr(#NotifyMsg,N_PRC_Err1)
        DEFAULT
      ENDSWITCH
;
    ;ENDFOLD (Advance)
;
    CASE #USR_TRIG
;
    ;FOLD Trig
;
      SWITCH FUNKTION
        CASE 523   ; Scanning stoppen
          N_PRC_MsgOff = 250
          B_PRC_MsgFlg = FALSE
          REPEAT
            N_PRC_Err1 = PRC_EndScan(nPAR4)
            N_PRC_Ret1 = PRC_MsgErr(#NotifyMsg,N_PRC_Err1)
          UNTIL (N_PRC_Ret1 == 1)
          IF B_PRC_MsgFlg THEN
            $FLAG[F_PRC_Err]   = TRUE
          ELSE
            $FLAG[F_PRC_NoErr] = TRUE
          ENDIF
        DEFAULT
      ENDSWITCH
;
    ;ENDFOLD (Trig)
;
    CASE #USR_MAIN
;
    ;FOLD Main
;
      PRC_MainPrg(FUNKTION,CMD_SEL,nPAR2,nPAR3,nPAR4,nPAR5,nPAR6,nPAR7,nPAR8)
;
    ;ENDFOLD (Main)
;
  ENDSWITCH
END
;
  ;ENDFOLD (Roboter Fuehrung)
;
  ;FOLD AutoGauge
;
GLOBAL DEF PRC_AutoGaugeInterface(USER_CMD:IN,CMD_SEL:IN,FUNKTION:IN,nPAR2:IN,nPAR3:IN,nPAR4:IN,nPAR5:IN,nPAR6:IN,nPAR7:IN,nPAR8:IN,nPAR9:IN)
DECL VW_USER_CMD USER_CMD
DECL INT         CMD_SEL
DECL INT         FUNKTION
DECL INT         nPAR2
DECL INT         nPAR3
DECL INT         nPAR4
DECL INT         nPAR5
DECL INT         nPAR6
DECL INT         nPAR7
DECL INT         nPAR8
DECL INT         nPAR9
DECL INT         nFlagCounter
  SWITCH USER_CMD
    CASE #USR_ADV
;
    ;FOLD Advance
;
      N_PRC_Err1   = 0
      N_PRC_Err2   = 0
      N_PRC_UpNr   = 0
      N_PRC_MsgOff = 0
      B_PRC_MsgFlg = FALSE
      FOR nFlagCounter = N_PRC_FiErr TO N_PRC_FiErr + N_PRC_LgErr
        $FLAG[nFlagCounter] = FALSE
      ENDFOR
      N_PRC_Err1 = PRC_CheckParams(nPAR2,nPAR3,nPAR4,nPAR5,nPAR6,nPAR7,nPAR8)
      IF N_PRC_Err1 > 0 THEN
        N_PRC_Ret1 = PRC_MsgErr(#DlgMsg,N_PRC_Err1)
        $FLAG[F_PRC_Err] = TRUE
        RETURN
      ENDIF
;
    ;ENDFOLD (Advance)
;
    CASE #USR_TRIG
;
    ;FOLD Trig
;
      RETURN
;
    ;ENDFOLD (Trig)
;
    CASE #USR_MAIN
;
    ;FOLD Main
;
      PRC_MainPrg(FUNKTION,CMD_SEL,nPAR2,nPAR3,nPAR4,nPAR5,nPAR6,nPAR7,nPAR8)
;
    ;ENDFOLD (Main)
;
  ENDSWITCH
END
;
  ;ENDFOLD (AutoGauge)
;
;ENDFOLD (Perceptron Interface)
;
;FOLD Perceptron Lokale Unterprogramme
;
  ;FOLD Messsystem initialisieren und Handshake synchronisieren
;
DEFFCT BOOL PRC_Sync()
INT nOutputCounter
INT nCounter1
INT nCounter2
  IF $IN[N_PRC_Ghost] THEN
    RETURN(TRUE)
  ENDIF
  B_PRC_ISTOOL = FALSE
  B_PRC_ISBASE = FALSE
  FOR nOutputCounter = 0 TO N_PRC_AnzWrt * 16
    $OUT[N_PRC_StrOut + nOutputCounter] = FALSE
  ENDFOR
  FOR nCounter1 = 1 to 17
    FOR nCounter2 = 1 to 6
      NA_PRC_Data[nCounter1,nCounter2] = 0
    ENDFOR
  ENDFOR
  B_PRC_InDone = FALSE   ; dadurch kein automatischer Reset Perceptron
  IF B_PRC_InDone THEN
    REPEAT
      N_PRC_Err1   = 1
      B_PRC_MsgFlg = FALSE
      N_PRC_Status = PRC_GetStatus()
      PRC_DebugDlg(1,N_PRC_Status,0)
      SWITCH N_PRC_Status
        CASE 50
          ; OK
        CASE 51,56,57,58,59,73,74,77,78,79,80,87,88,93
          B_PRC_MsgFlg = TRUE
        DEFAULT
          N_PRC_Status = 59
          B_PRC_MsgFlg = TRUE
      ENDSWITCH
      IF B_PRC_MsgFlg THEN
        B_PRC_MsgKri = TRUE
        N_PRC_Ret1   = PRC_MsgErr(#NotifyMsg,N_PRC_Status)
      ENDIF
      IF N_PRC_Status <> 50 THEN
        B_PRC_MsgKri = TRUE
        N_PRC_Ret1 = PRC_MsgErr(#NotifyMsg,95)
        IF N_PRC_Ret1 == 2 THEN
          REPEAT
            PRC_DebugDlg(9,0,0)
            N_PRC_Err2 = PRC_Reset()
            B_PRC_MsgKri = TRUE
            N_PRC_Ret2 = PRC_MsgErr(#NotifyMsg,N_PRC_Err2)
          UNTIL (N_PRC_Ret2 == 1)
        ENDIF
      ELSE
        N_PRC_Ret1 = PRC_MsgErr(#NotifyMsg,N_PRC_Status)
      ENDIF
    UNTIL (N_PRC_Ret1 == 1)
    IF (B_PRC_MsgFlg == TRUE) THEN
      $FLAG[F_PRC_Err]   = TRUE
      $FLAG[F_PRC_NoErr] = FALSE
    ELSE
      $FLAG[F_PRC_Err]   = FALSE
      $FLAG[F_PRC_NoErr] = TRUE
    ENDIF
    B_PRC_InDone = TRUE
  ENDIF
;
  GLOBAL INTERRUPT DECL N_PRC_Int1 WHEN $OUT[N_PRC_RobMv]   DO PRC_Move(1)
  GLOBAL INTERRUPT DECL N_PRC_Int2 WHEN $OUT[N_PRC_RobNoMv] DO PRC_Move(2)
  INTERRUPT ON N_PRC_Int1
  INTERRUPT ON N_PRC_Int2
;
  RETURN(TRUE)
ENDFCT
;
  ;ENDFOLD (Messsystem initialisieren und Handshake synchronisieren)
;
  ;FOLD Main Programm
;
GLOBAL DEF PRC_MainPrg(FUNKTION:IN,CMD_SEL:IN,nPAR2:IN,nPAR3:IN,nPAR4:IN,nPAR5:IN,nPAR6:IN,nPAR7:IN,nPAR8:IN)
INT FUNKTION
INT CMD_SEL
INT nPAR2
INT nPAR3
INT nPAR4
INT nPAR5
INT nPAR6
INT nPAR7
INT nPAR8
INT I
  N_PRC_PktNr = nPAR4
  N_PRC_BasNr = $ACT_BASE
  N_PRC_TooNr = $ACT_TOOL
  B_PRC_Ghost = $IN[N_PRC_Ghost]
  ; bei Geisterschicht nur Messung starten, da
  ; dabei auch UP mit Punktmessung gestartet wird
  IF ((B_PRC_Ghost) AND (FUNKTION <> 510)) THEN
    $FLAG[F_PRC_Err]   = FALSE
    $FLAG[F_PRC_NoErr] = TRUE
    RETURN
  ENDIF
  SWITCH FUNKTION
    CASE 501 ; Statusanforderung
      N_PRC_MsgOff   = 300
      REPEAT
        N_PRC_Err1   = 1
        B_PRC_MsgFlg = FALSE
        N_PRC_Status = PRC_GetStatus()
        PRC_DebugDlg(1,N_PRC_Status,0)
        SWITCH N_PRC_Status
          CASE 300
            ; OK
          CASE 301,306,307,308,309,317,318,323,324,327,328,329,330,343
            B_PRC_MsgFlg = TRUE
          DEFAULT
            N_PRC_Status = 309
            B_PRC_MsgFlg = TRUE
        ENDSWITCH
        IF B_PRC_MsgFlg THEN
          N_PRC_Ret1 = PRC_MsgErr(#NotifyMsg,N_PRC_Status)
        ENDIF
        IF N_PRC_Status <> 300 THEN
          N_PRC_Ret1 = PRC_MsgErr(#NotifyMsg,345)
          IF N_PRC_Ret1 == 2 THEN
            REPEAT
              PRC_DebugDlg(9,0,0)
              N_PRC_Err2 = PRC_Reset()
              N_PRC_Ret2 = PRC_MsgErr(#NotifyMsg,N_PRC_Err2)
            UNTIL (N_PRC_Ret2 == 1)
          ENDIF
        ELSE
          N_PRC_Ret1 = PRC_MsgErr(#NotifyMsg,1,N_PRC_Status)
        ENDIF
      UNTIL (N_PRC_Ret1 == 1)
      IF (B_PRC_MsgFlg == TRUE) THEN
        $FLAG[F_PRC_Err]   = TRUE
        $FLAG[F_PRC_NoErr] = FALSE
      ELSE
        $FLAG[F_PRC_Err]   = FALSE
        $FLAG[F_PRC_NoErr] = TRUE
      ENDIF
    CASE 510,514 ; Messung mit Punktmessung starten
      N_PRC_MsgOff = 100
      B_PRC_MsgFlg = FALSE
      SWITCH CMD_SEL
        CASE 1001 ;IMT  ; Hauptgruppe 9, Untergruppe 1
          IF (FUNKTION == 514) THEN
            O_PRC_CmpStr = TRUE
          ENDIF
          REPEAT
            N_PRC_Err1   = 0
            B_PRC_MsgFlg = FALSE
            PRC_DebugDlg(6,0,0)
            PRC_DebugDlg(25,nPAR2,nPAR3)
            PRC_StartMessung(nPAR2,nPAR3,nPAR6)
            SWITCH N_PRC_Err1
              CASE 100
                ; OK
              CASE 105,106,107,108,109,111,112,143
                B_PRC_MsgFlg = TRUE
              DEFAULT
                B_PRC_MsgFlg = TRUE
            ENDSWITCH
            N_PRC_Ret1 = PRC_MsgErr(#NotifyMsg,N_PRC_Err1)
            IF N_PRC_Ret1 == 2 THEN
              N_PRC_MsgOff = 100
              REPEAT
                PRC_DebugDlg(9,0,0)
                N_PRC_Err2 = PRC_Reset()
                N_PRC_Ret2 = PRC_MsgErr(#NotifyMsg,N_PRC_Err2)
              UNTIL (N_PRC_Ret2 == 1)
            ENDIF
          UNTIL (N_PRC_Ret1 == 1)
          IF (B_PRC_MsgFlg) THEN
            $FLAG[F_PRC_Err]   = TRUE
          ELSE
            $FLAG[F_PRC_NoErr] = TRUE
          ENDIF
          O_PRC_CmpStr = FALSE
        CASE 1003 ;AutoGauge  ; Hauptgruppe 9, Untergruppe 3
          N_PRC_Ret1 = PRC_MsgErr(#NotifyMsg,910,FUNKTION,CMD_SEL)
        DEFAULT
          N_PRC_Ret1 = PRC_MsgErr(#NotifyMsg,910,FUNKTION,CMD_SEL)
      ENDSWITCH
    CASE 511 ; Mess UP-Nummer holen fuer Punktmessung
      N_PRC_MsgOff = 800
      B_PRC_MsgFlg = FALSE
      SWITCH CMD_SEL
        CASE 1002 ; RF  ; Hauptgruppe 9, Untergruppe 1 + 2
          PRC_DebugDlg(24,0,0)
          N_PRC_Ret1 = PRC_GetMessUpNr(nPAR2,nPAR3,nPAR6)
          SWITCH N_PRC_Ret1
            CASE 800
              ; OK
            CASE 801,807,829,840,841
              $FLAG[F_PRC_Err] = TRUE
              B_PRC_MsgFlg     = TRUE
            DEFAULT
              $FLAG[F_PRC_Err] = TRUE
              B_PRC_MsgFlg     = TRUE
          ENDSWITCH
        CASE 1003 ; AutoGauge  ; Hauptgruppe 9, Untergruppe 3
         N_PRC_Ret1 = PRC_MsgErr(#NotifyMsg,910,FUNKTION,CMD_SEL)
        DEFAULT
          N_PRC_Ret1 = PRC_MsgErr(#NotifyMsg,910,FUNKTION,CMD_SEL)
      ENDSWITCH
    CASE 512 ; Kompensations UP-Nummer holen fuer Punktmessung
      N_PRC_MsgOff = 800
      B_PRC_MsgFlg = FALSE
      SWITCH CMD_SEL
        CASE 1002 ; RF  ; Hauptgruppe 9, Untergruppe 1 + 2
          PRC_DebugDlg(24,0,0)
          N_PRC_Ret1 = PRC_GetKompUpNr(nPAR2,nPAR3,nPAR6)
          SWITCH N_PRC_Ret1
            CASE 800,850,851,852,853,860,861
              ; OK
            CASE 801,807,809,811,829,840,841,843,870,871
              $FLAG[F_PRC_Err] = TRUE
              B_PRC_MsgFlg     = TRUE
            DEFAULT
              $FLAG[F_PRC_Err] = TRUE
              B_PRC_MsgFlg     = TRUE
          ENDSWITCH
        CASE 1003 ; AutoGauge  ; Hauptgruppe 9, Untergruppe 3
          N_PRC_Ret1 = PRC_MsgErr(#NotifyMsg,910,FUNKTION,CMD_SEL)
        DEFAULT
          N_PRC_Ret1 = PRC_MsgErr(#NotifyMsg,910,FUNKTION,CMD_SEL)
      ENDSWITCH
    CASE 513 ; Messen komplett
      N_PRC_MsgOff = 100
      B_PRC_MsgFlg = FALSE
      SWITCH CMD_SEL
        CASE 1002,1003 ; RF / AG ; Hauptgruppe 9, Untergruppe 2 + 3
          REPEAT
            N_PRC_Err1   = 0
            B_PRC_MsgFlg = FALSE
            PRC_DebugDlg(6,0,0)
            PRC_DebugDlg(25,nPAR2,nPAR3)
            PRC_StartMessung(nPAR2,nPAR3,nPAR6)
            SWITCH N_PRC_Err1
              CASE 100
                ; OK
              CASE 105,106,107,108,109,111,112,143
                B_PRC_MsgFlg = TRUE
              DEFAULT
                B_PRC_MsgFlg = TRUE
            ENDSWITCH
            N_PRC_Ret1 = PRC_MsgErr(#NotifyMsg,N_PRC_Err1)
            IF N_PRC_Ret1 == 2 THEN
              N_PRC_MsgOff = 100
              REPEAT
                PRC_DebugDlg(9,0,0)
                N_PRC_Err2 = PRC_Reset()
                N_PRC_Ret2 = PRC_MsgErr(#NotifyMsg,N_PRC_Err2)
              UNTIL (N_PRC_Ret2 == 1)
            ENDIF
          UNTIL (N_PRC_Ret1 == 1)
          IF (B_PRC_MsgFlg) THEN
            $FLAG[F_PRC_Err]   = TRUE
          ELSE
            $FLAG[F_PRC_NoErr] = TRUE
          ENDIF
          N_PRC_MsgOff = 400
          B_PRC_MsgFlg = FALSE
          N_PRC_Err1   =  1
          IF (FUNKTION == 530) THEN
            PRC_DebugDlg(4,0,0)
            PRC_MessungBeenden(CMD_SEL)
          ENDIF
          N_PRC_Ret1 = PRC_MsgErr(#NotifyMsg,N_PRC_Err1)
          IF B_PRC_MsgFlg THEN
            $FLAG[F_PRC_Err]   = TRUE
          ELSE
            $FLAG[F_PRC_NoErr] = TRUE
          ENDIF
        DEFAULT
          N_PRC_Ret1 = PRC_MsgErr(#NotifyMsg,910,FUNKTION,CMD_SEL)
      ENDSWITCH
    CASE 520 ;Punktmessung starten
      N_PRC_MsgOff = 200
      B_PRC_MsgFlg = FALSE
      SWITCH CMD_SEL
        CASE 1002 ; RF  ; Hauptgruppe 9, Untergruppe 2
          N_PRC_Ret1 = PRC_MsgErr(#NotifyMsg,910,FUNKTION,CMD_SEL)
        CASE 1003 ;AutoGauge  ; Hauptgruppe 9, Untergruppe 3
          N_PRC_Ret1 = PRC_MsgErr(#NotifyMsg,910,FUNKTION,CMD_SEL)
        DEFAULT
          N_PRC_Ret1 = PRC_MsgErr(#NotifyMsg,910,FUNKTION,CMD_SEL)
      ENDSWITCH
    CASE 521 ; Punkte beendet
      N_PRC_MsgOff = 200
      B_PRC_MsgFlg = FALSE
      SWITCH CMD_SEL
        CASE 1002 ; RF  ; Hauptgruppe 9, Untergruppe 1 + 2
          REPEAT
            PRC_DebugDlg(3,N_PRC_LstPkt,0)
            PRC_PunktMessung(N_PRC_LstPkt,-1,-1)
            N_PRC_Ret1 = PRC_MsgErr(#NotifyMsg,N_PRC_Err1,0,N_PRC_LstPkt)
          UNTIL (N_PRC_Ret1 == 1)
          IF B_PRC_MsgFlg THEN
            $FLAG[F_PRC_Err]   = TRUE
          ELSE
            $FLAG[F_PRC_NoErr] = TRUE
          ENDIF
        CASE 1003 ; AG  ; Hauptgruppe 9, Untergruppe 3
          N_PRC_Ret1 = PRC_MsgErr(#NotifyMsg,910,FUNKTION,CMD_SEL)
        DEFAULT
          N_PRC_Ret1 = PRC_MsgErr(#NotifyMsg,910,FUNKTION,CMD_SEL)
      ENDSWITCH
    CASE 522 ;Scanning starten
      N_PRC_MsgOff = 250
      B_PRC_MsgFlg = FALSE
      SWITCH CMD_SEL
        CASE 1002 ; RF  ; Hauptgruppe 9, Untergruppe 2
          N_PRC_Ret1 = PRC_MsgErr(#NotifyMsg,910,FUNKTION,CMD_SEL)
        CASE 1003 ;AutoGauge  ; Hauptgruppe 9, Untergruppe 3
          N_PRC_Ret1 = PRC_MsgErr(#NotifyMsg,910,FUNKTION,CMD_SEL)
        DEFAULT
          N_PRC_Ret1 = PRC_MsgErr(#NotifyMsg,910,FUNKTION,CMD_SEL)
      ENDSWITCH
    CASE 523
    ; in TRIG ausgelagert
	CASE 525 ; Sende Pose_ID
      N_PRC_MsgOff = 200
      B_PRC_MsgFlg = FALSE
      SWITCH CMD_SEL
        CASE 1002 ; RF  ; Hauptgruppe 9, Untergruppe 2
          N_PRC_Ret1 = PRC_MsgErr(#NotifyMsg,910,FUNKTION,CMD_SEL)
        CASE 1003 ;AutoGauge  ; Hauptgruppe 9, Untergruppe 3
          N_PRC_Ret1 = PRC_MsgErr(#NotifyMsg,910,FUNKTION,CMD_SEL)
        DEFAULT
          N_PRC_Ret1 = PRC_MsgErr(#NotifyMsg,910,FUNKTION,CMD_SEL)
      ENDSWITCH
    CASE 530 ;Messung beenden
      N_PRC_MsgOff = 400
      B_PRC_MsgFlg = FALSE
      SWITCH CMD_SEL
        CASE 1002 ; RF ; Hauptgruppe 9, Untergruppe 1 + 2
          N_PRC_Err1   =  1
            PRC_DebugDlg(4,0,0)
            PRC_MessungBeenden(CMD_SEL)
          N_PRC_Ret1 = PRC_MsgErr(#NotifyMsg,N_PRC_Err1)
          IF B_PRC_MsgFlg THEN
            $FLAG[F_PRC_Err]   = TRUE
          ELSE
            $FLAG[F_PRC_NoErr] = TRUE
          ENDIF
        CASE 1003 ;AutoGauge  ; Hauptgruppe 9, Untergruppe 3
          N_PRC_Ret1 = PRC_MsgErr(#NotifyMsg,910,FUNKTION,CMD_SEL)
        DEFAULT
          N_PRC_Ret1=PRC_MsgErr(#NotifyMsg,910,FUNKTION,CMD_SEL)
      ENDSWITCH
    CASE 540 ;Sensortausch (Messung mit Punktmessung)
      PRC_DebugDlg(5,0,0)
      N_PRC_MsgOff = 600
      B_PRC_MsgFlg = FALSE
      B_PRC_1Kalib = FALSE
      B_PRC_TmpKalib = FALSE
      B_PRC_ToFiOK=FALSE
      SWITCH CMD_SEL
        CASE 1002 ; RF  ; Hauptgruppe 9, Untergruppe 1 + 2
          IF (($mode_op <> #T1) AND ($mode_op <> #T2)) THEN
            N_PRC_Err1   = 639
            B_PRC_MsgFlg = TRUE
            N_PRC_Ret1   = PRC_MsgErr(#NotifyMsg,N_PRC_Err1)
            $FLAG[F_PRC_Err] = TRUE
            RETURN
          ENDIF
          LOOP
            REPEAT ; Sensorpruefung
              N_PRC_ModNr = N_PRC_SenPrM
              N_PRC_UpNr  = N_PRC_SenPrU
              REPEAT
                N_PRC_Err1   = 0
                N_PRC_Ret1   = 1
                B_PRC_MsgFlg = FALSE
                N_PRC_Status = PRC_GetStatus()
                PRC_DebugDlg(1,N_PRC_Status,0)
                IF B_PRC_MsgFlg THEN
                  N_PRC_Ret1 = PRC_MsgErr(#NotifyMsg,N_PRC_Status)
                  RETURN
                ELSE
                  IF (N_PRC_Status <> 600) THEN
                    N_PRC_Status=606
                    N_PRC_Ret1   = PRC_MsgErr(#NotifyMsg,N_PRC_Status)
                    SWITCH N_PRC_Ret1
                    CASE 1
                      N_PRC_Ret1   = PRC_MsgErr(#NotifyMsg,644)
                      return
                    CASE 2
                      N_PRC_Ret1   = 0
                    DEFAULT
                      ;falsche Dialogantwort
                      $FLAG[F_PRC_Err]   = TRUE
                      RETURN
                    ENDSWITCH
                  ELSE
                    N_PRC_Ret1 = 1
                  ENDIF
                ENDIF
              UNTIL (N_PRC_Ret1 == 1)
              IF B_PRC_MsgFlg THEN
                $FLAG[F_PRC_Err] = TRUE
                RETURN
              ENDIF
              B_PRC_ISTOOL = TRUE
              PRC_DebugDlg(16,0,0)
              PRC_DebugDlg(25,N_PRC_ModNr,N_PRC_UpNr)
              N_PRC_MsrErg = PRC_StartMsrPktMsr(N_PRC_ModNr,N_PRC_UpNr,nPAR6)
              N_PRC_MsgOff = 600
              IF B_PRC_MsgFlg THEN
                B_PRC_ISTOOL = FALSE
                $FLAG[F_PRC_Err] = TRUE
                RETURN
              ENDIF
              SWITCH N_PRC_MsrErg
                CASE 600,601  ;alles ok
                  N_PRC_Ret1 = PRC_MsgErr(#NotifyMsg,633)
                  B_PRC_ISTOOL = FALSE
                  if B_PRC_1Kalib then ;min 1mal kalib
                     B_PRC_ToFiOK=TRUE
                     if ((N_PRC_SubSystem == 1) and not B_PRC_TmpKalib) then
                        ;Tempkalib ausfuehren
                     else
                       N_PRC_Ret1 = PRC_MsgErr(#NotifyMsg,698)
                       $FLAG[F_PRC_NoErr] = TRUE
                       RETURN
                    endif
                  endif
                CASE 1151, 1152, 1155, 1156   ; Kalibrierung erforderlich
                  N_PRC_RET1 = 1
                CASE 603, 605, 606, 607, 1153, 1154, 1157, 1158   ; Sensormontage pruefen
                  N_PRC_MsrErg = 610
                  N_PRC_Ret1   = PRC_MsgErr(#NotifyMsg,N_PRC_MsrErg)
                  IF N_PRC_Ret1 == 1 THEN
                    B_PRC_ISTOOL = FALSE
                    $FLAG[F_PRC_Err] = TRUE
                    RETURN
                  ENDIF
                DEFAULT
                  N_PRC_Ret1 = PRC_MsgErr(#NotifyMsg,N_PRC_Err1)
                  B_PRC_ISTOOL = FALSE
                  $FLAG[F_PRC_Err] = TRUE
                  RETURN
              ENDSWITCH
            UNTIL N_PRC_Ret1 == 1
            B_PRC_ISTOOL = FALSE
            if (((N_PRC_SubSystem == 1) and (B_PRC_ToFiOK)) OR (N_PRC_SubSystem == 0))then
              N_PRC_Ret1   = PRC_MsgErr(#NotifyMsg,630)
            else
              N_PRC_Ret1   = PRC_MsgErr(#NotifyMsg,650)
            endif
            REPEAT
              N_PRC_Err1   = 0
              B_PRC_MsgFlg = FALSE
              N_PRC_Status = PRC_GetStatus()
              PRC_DebugDlg(1,N_PRC_Status,0)
              IF ((N_PRC_SubSystem == 1) AND NOT(B_PRC_ToFiOK)) THEN
                 if (N_PRC_Status <> 630) then
                   N_PRC_Err1   = 652   ; Perceptron nicht in Toolfinder-Modus
                   B_PRC_MsgFlg = TRUE
                endif
              endif
              IF ((N_PRC_SubSystem <> 1) OR ((N_PRC_SubSystem == 1) AND (B_PRC_ToFiOK))) then
                if(N_PRC_Status <> 623) THEN
                   N_PRC_Err1   = 632   ; Perceptron nicht in Kalibrier-Modus
                   B_PRC_MsgFlg = TRUE
                endif
              endif
              IF B_PRC_MsgFlg THEN
                N_PRC_Ret1 = PRC_MsgErr(#NotifyMsg,N_PRC_Err1)
              ELSE
                N_PRC_Ret1   = 1
              ENDIF
            UNTIL (N_PRC_Ret1 == 1)
            IF (B_PRC_MsgFlg) THEN
              $FLAG[F_PRC_Err] = TRUE
              RETURN
            ENDIF
            IF (((N_PRC_SubSystem == 1) and B_PRC_ToFiOK) OR (N_PRC_SubSystem == 0)) then
              N_PRC_ModNr = N_PRC_TmpCmpM
              N_PRC_UpNr  = N_PRC_TmpCmpU
              B_PRC_TmpKalib = TRUE
            else
              N_PRC_ModNr = N_PRC_SenTaM
              N_PRC_UpNr  = N_PRC_SenTaU
            endif
            PRC_DebugDlg(26,0,0)
            PRC_DebugDlg(25,N_PRC_ModNr,N_PRC_UpNr)
            N_PRC_MsrErg = PRC_StartMsrPktMsr(N_PRC_ModNr,N_PRC_UpNr,nPAR6) ; Starten im Toolfinder od. Kalib-Modus
            N_PRC_MsgOff = 600
            IF B_PRC_MsgFlg THEN
              N_PRC_Ret1       = PRC_MsgErr(#NotifyMsg,N_PRC_Err1)
              $FLAG[F_PRC_Err] = TRUE
              RETURN
            ENDIF
            IF (((N_PRC_SubSystem == 1) and B_PRC_ToFiOK)  OR (N_PRC_SubSystem == 0)) then
              N_PRC_Ret1 = PRC_MsgErr(#NotifyMsg,699)
            ELSE
              N_PRC_Ret1 = PRC_MsgErr(#NotifyMsg,653)
            ENDIF
            B_PRC_1Kalib = TRUE
          ENDLOOP
        CASE 1003 ;AutoGauge  ; Hauptgruppe 9, Untergruppe 3
          N_PRC_Ret1 = PRC_MsgErr(#NotifyMsg,910,FUNKTION,CMD_SEL)
        DEFAULT
          N_PRC_Ret1=PRC_MsgErr(#NotifyMsg,910,FUNKTION,CMD_SEL)
      ENDSWITCH
    CASE 545 ;Robotertausch
      PRC_DebugDlg(10,0,0)
      N_PRC_MsgOff   = 700
      B_PRC_MsgFlg   = FALSE
      B_PRC_TmpKalib = FALSE
      B_PRC_ToFiOK   = FALSE
      B_PRC_NoBaKo   = FALSE
      SWITCH CMD_SEL
        CASE 1002 ; RF  ; Hauptgruppe 9, Untergruppe 1 + 2
          IF (($mode_op <> #T1) AND ($mode_op <> #T2)) THEN
            N_PRC_Err1 = 739
            B_PRC_MsgFlg = TRUE
            N_PRC_Ret1 = PRC_MsgErr(#NotifyMsg,N_PRC_Err1)
            $FLAG[F_PRC_Err] = TRUE
            RETURN
          ENDIF
          REPEAT ; Roboterpruefung
            N_PRC_ModNr = N_PRC_RobPrM
            N_PRC_UpNr  = N_PRC_RobPrU
            REPEAT
              N_PRC_Err1   = 0
              N_PRC_Ret1   = 1
              B_PRC_MsgFlg = FALSE
              N_PRC_Status = PRC_GetStatus()
              PRC_DebugDlg(1,N_PRC_Status,0)
              IF B_PRC_MsgFlg THEN
                N_PRC_Ret1 = PRC_MsgErr(#NotifyMsg,N_PRC_Status)
                RETURN
              ELSE
                IF (N_PRC_Status <> 700) THEN
                  N_PRC_Ret1   = PRC_MsgErr(#NotifyMsg,N_PRC_Status)
                  SWITCH N_PRC_Ret1
                  CASE 1
                    N_PRC_Ret1   = PRC_MsgErr(#NotifyMsg,744)
                    RETURN
                  CASE 2
                    N_PRC_Ret1   = 0
                  DEFAULT
                    ;falsche Dialogantwort
                    $FLAG[F_PRC_Err]   = TRUE
                    RETURN
                  ENDSWITCH
                ELSE
                  N_PRC_Ret1 = 1
                ENDIF
              ENDIF
            UNTIL(N_PRC_Ret1 == 1)
            IF B_PRC_MsgFlg THEN
              $FLAG[F_PRC_Err] = TRUE
              RETURN
            ENDIF
            B_PRC_ISBASE = TRUE
            PRC_DebugDlg(6,0,0)
            PRC_DebugDlg(25,N_PRC_ModNr,N_PRC_UpNr)
            N_PRC_MsrErg = PRC_StartMsrPktMsr(N_PRC_ModNr,N_PRC_UpNr,nPAR6)
            N_PRC_MsgOff = 700
            IF B_PRC_MsgFlg THEN
              B_PRC_ISBASE = FALSE
              $FLAG[F_PRC_Err] = TRUE
              RETURN
            ENDIF
            SWITCH N_PRC_MsrErg
              CASE 700, 1152, 1156; alles ok. ,Sensortoleranz
                if (N_PRC_MsrErg == 700) then
                  ;N_PRC_Ret1 = PRC_MsgErr(#NotifyMsg,733)
                endif
                B_PRC_ISBASE = FALSE
                ;---------Sensortausch -----------------------------
                PRC_DebugDlg(5,0,0)
                N_PRC_MsgOff = 600
                B_PRC_MsgFlg = FALSE
                B_SensIsKalib = FALSE
                IF (($mode_op <> #T1) AND ($mode_op <> #T2)) THEN
                  N_PRC_Err1   = 639
                  B_PRC_MsgFlg = TRUE
                  N_PRC_Ret1   = PRC_MsgErr(#NotifyMsg,N_PRC_Err1)
                  $FLAG[F_PRC_Err] = TRUE
                  RETURN
                ENDIF
                Repeat
                  ;-------------Sensorkalibrierung-------------------
                  B_PRC_ISTOOL = FALSE
                  IF (N_PRC_SubSystem==1) THEN
                    N_PRC_Ret1   = PRC_MsgErr(#NotifyMsg,650)
                  ELSE
                    N_PRC_Ret1   = PRC_MsgErr(#NotifyMsg,630)
                  ENDIF
                  REPEAT
                    N_PRC_Err1   = 0
                    B_PRC_MsgFlg = FALSE
                    N_PRC_Status = PRC_GetStatus()
                    PRC_DebugDlg(1,N_PRC_Status,0)
                    IF (N_PRC_SubSystem == 1) THEN
                      if (N_PRC_Status <> 630) then
                        N_PRC_Err1   = 652   ; Perceptron nicht in Toolfinder-Modus
                        B_PRC_MsgFlg = TRUE
                      endif
                    endif
                    IF (N_PRC_SubSystem <> 1) then
                      if(N_PRC_Status <> 623) THEN
                        N_PRC_Err1   = 632   ; Perceptron nicht in Kalibrier-Modus
                        B_PRC_MsgFlg = TRUE
                      endif
                    endif
                    IF B_PRC_MsgFlg THEN
                      N_PRC_Ret1 = PRC_MsgErr(#NotifyMsg,N_PRC_Err1)
                    ELSE
                      N_PRC_Ret1   = 1
                    ENDIF
                  UNTIL (N_PRC_Ret1 == 1)
                  IF (B_PRC_MsgFlg) THEN
                    $FLAG[F_PRC_Err] = TRUE
                    RETURN
                  ENDIF
                  IF (N_PRC_SubSystem == 1) then
                    N_PRC_ModNr = N_PRC_SenTaM
                    N_PRC_UpNr  = N_PRC_SenTaU
                  else
                    N_PRC_ModNr = N_PRC_TmpCmpM
                    N_PRC_UpNr  = N_PRC_TmpCmpU
                  endif
                  PRC_DebugDlg(26,0,0)
                  PRC_DebugDlg(25,N_PRC_ModNr,N_PRC_UpNr)
                  N_PRC_MsrErg = PRC_StartMsrPktMsr(N_PRC_ModNr,N_PRC_UpNr,nPAR6) ; Starten im Toolfinder-Modus
                  N_PRC_MsgOff = 600
                  IF B_PRC_MsgFlg THEN
                    N_PRC_Ret1       = PRC_MsgErr(#NotifyMsg,N_PRC_Err1)
                    $FLAG[F_PRC_Err] = TRUE
                    RETURN
                  ENDIF
                  SWITCH N_PRC_MsrErg
                    CASE 600,601  ;alles ok
                      ;N_PRC_Ret1 = PRC_MsgErr(#NotifyMsg,699)
                      $FLAG[F_PRC_NoErr] = TRUE
                      B_SensIsKalib = TRUE
                    CASE 1151, 1152, 1155, 1156   ; Kalibrierung erforderlich
                      N_PRC_RET1 = 1
                    CASE 603, 605, 606, 607, 1153, 1154, 1157, 1158   ; Sensormontage pruefen
                      N_PRC_MsrErg = 610
                      N_PRC_Ret1   = PRC_MsgErr(#NotifyMsg,N_PRC_MsrErg)
                      IF N_PRC_Ret1 == 1 THEN
                        B_PRC_ISTOOL = FALSE
                        $FLAG[F_PRC_Err] = TRUE
                        RETURN
                      ENDIF
                    DEFAULT
                      N_PRC_Ret1 = PRC_MsgErr(#NotifyMsg,N_PRC_Err1)
                      B_PRC_ISTOOL = FALSE
                      $FLAG[F_PRC_Err] = TRUE
                      RETURN
                  ENDSWITCH
                Until B_SensIsKalib
                IF (N_PRC_SubSystem == 1) then
                  N_PRC_Ret1 = PRC_MsgErr(#NotifyMsg,796)
                else
;                 N_PRC_Ret1 = PRC_MsgErr(#NotifyMsg,699)
                ENDIF
                ;---------------ende Sensorkalibrierung-------------------
                N_PRC_MsgOff = 700
                B_PRC_MsgFlg = FALSE
              CASE 703, 705, 706, 707, 1151, 1152, 1153, 1154, 1155, 1157, 1158   ;Robotermontage pruefen
                N_PRC_MsrErg = 710
                N_PRC_Ret1 = PRC_MsgErr(#NotifyMsg,N_PRC_MsrErg)
                IF N_PRC_Ret1 == 1 THEN
                  B_PRC_ISBASE = FALSE
                  $FLAG[F_PRC_Err] = TRUE
                  RETURN
                ENDIF
              DEFAULT
                B_PRC_ISBASE = FALSE
                N_PRC_Ret1 = PRC_MsgErr(#NotifyMsg,N_PRC_Err1)
                $FLAG[F_PRC_Err] = TRUE
                RETURN
            ENDSWITCH
          UNTIL (N_PRC_Ret1 == 1)
          B_PRC_ISBASE = FALSE
          REPEAT
            REPEAT
              N_PRC_MsgOff = 700
              N_PRC_Err1   = PRC_MsgErr(#NotifyMsg,730)
              N_PRC_Err1   = 0
              B_PRC_MsgFlg = FALSE
              N_PRC_Status = PRC_GetStatus()
              PRC_DebugDlg(1,N_PRC_Status,0)
              IF (N_PRC_Status <> 700) THEN
                N_PRC_Err1   = 732 ; Perceptron nicht in Automtikmodus
                B_PRC_MsgFlg = TRUE
              ELSE
                B_PRC_MsgFlg = FALSE
                N_PRC_Ret1   = 1
              ENDIF
              IF B_PRC_MsgFlg THEN
                N_PRC_Ret1 = PRC_MsgErr(#NotifyMsg,N_PRC_Err1)
              ENDIF
            UNTIL (N_PRC_Ret1 == 1)
            IF (B_PRC_MsgFlg) THEN
              $FLAG[F_PRC_Err] = TRUE
              RETURN
            ENDIF
            N_PRC_ModNr  = N_PRC_RobTaM
            N_PRC_UpNr   = N_PRC_RobTaU
            PRC_DebugDlg(6,0,0)
            PRC_DebugDlg(25,N_PRC_ModNr,N_PRC_UpNr)
            N_PRC_MsrErg = PRC_StartMsrPktMsr(N_PRC_ModNr,N_PRC_UpNr,nPAR6)
            N_PRC_MsgOff = 700
            IF B_PRC_MsgFlg THEN
              N_PRC_Ret1 = PRC_MsgErr(#NotifyMsg,N_PRC_Err1)
              $FLAG[F_PRC_Err] = TRUE
              RETURN
            ENDIF
            SWITCH N_PRC_MsrErg
              CASE 700,701  ;alles ok
                ;N_PRC_Ret1 = PRC_MsgErr(#NotifyMsg,733)
                IF ((N_PRC_Subsystem == 1) and NOT(B_PRC_TMPKALIB)) THEN
                    ;-------------Sensorkalibrierung-------------------
                  B_SensIsKalib = FALSE
                  N_PRC_MsgOff = 600
                  N_PRC_Ret1   = PRC_MsgErr(#NotifyMsg,795)
                  Repeat
                    B_PRC_ISTOOL = FALSE
                    N_PRC_Ret1   = PRC_MsgErr(#NotifyMsg,630)
                    REPEAT
                      N_PRC_Err1   = 0
                      B_PRC_MsgFlg = FALSE
                      N_PRC_Status = PRC_GetStatus()
                      PRC_DebugDlg(1,N_PRC_Status,0)
                      IF (N_PRC_Status <> 623) THEN ;kalibmode
                        N_PRC_Err1   = 632   ; Perceptron nicht in Kalibrier-Modus
                        B_PRC_MsgFlg = TRUE
                      ELSE
                        B_PRC_MsgFlg = FALSE
                        N_PRC_Ret1   = 1
                      ENDIF
                      IF B_PRC_MsgFlg THEN
                       N_PRC_Ret1 = PRC_MsgErr(#NotifyMsg,N_PRC_Err1)
                      ENDIF
                    UNTIL (N_PRC_Ret1 == 1)
                    IF (B_PRC_MsgFlg) THEN
                      $FLAG[F_PRC_Err] = TRUE
                      RETURN
                    ENDIF
                    N_PRC_ModNr = N_PRC_TmpCmpM
                    N_PRC_UpNr  = N_PRC_TmpCmpU
                    PRC_DebugDlg(26,0,0)
                    PRC_DebugDlg(25,N_PRC_ModNr,N_PRC_UpNr)
                    N_PRC_MsrErg = PRC_StartMsrPktMsr(N_PRC_ModNr,N_PRC_UpNr,nPAR6) ; Starten im Kalibrier-Modus
                    N_PRC_MsgOff = 600
                    IF B_PRC_MsgFlg THEN
                      N_PRC_Ret1       = PRC_MsgErr(#NotifyMsg,N_PRC_Err1)
                      $FLAG[F_PRC_Err] = TRUE
                      RETURN
                    ENDIF
                    SWITCH N_PRC_MsrErg
                      CASE 600,601  ;alles ok
                        ;N_PRC_Ret1 = PRC_MsgErr(#NotifyMsg,699)
                        $FLAG[F_PRC_NoErr] = TRUE
                        B_SensIsKalib = TRUE
                        B_PRC_TmpKalib = TRUE
                      CASE 1152, 1156   ; Kalibrierung erforderlich
                        N_PRC_RET1 = 1
                      CASE 1153, 1154, 1157, 1158   ; Sensormontage pruefen
                        N_PRC_MsrErg = 610
                        N_PRC_Ret1   = PRC_MsgErr(#NotifyMsg,N_PRC_MsrErg)
                        IF N_PRC_Ret1 == 1 THEN
                          B_PRC_ISTOOL = FALSE
                          $FLAG[F_PRC_Err] = TRUE
                          RETURN
                        ENDIF
                      DEFAULT
                        N_PRC_Ret1 = PRC_MsgErr(#NotifyMsg,N_PRC_Err1)
                        B_PRC_ISTOOL = FALSE
                        $FLAG[F_PRC_Err] = TRUE
                        RETURN
                    ENDSWITCH
                  Until B_SensIsKalib
                  ;---------------ende Sensorkalibrierung-------------------
                ENDIF
                B_PRC_ISBase = FALSE
                IF not(B_PRC_NoBaKo) then
                  N_PRC_RET1   = 0
                  B_PRC_NoBaKo = TRUE
                else
                  N_PRC_RET1 = 1
                endif
              CASE 1151, 1152, 1155, 1156   ; Korrektur holen+aufrechnen
                N_PRC_Ret1 = PRC_MsgErr(#NotifyMsg,797)
                VF_PRC_RobKor = $BASE:AVF_PRC_Korr[N_PRC_VFNr]:INV_POS($BASE)
                ;halt ; VF_PRC_RobKor checken
                FOR I = 1 TO MAX_BASE
                  BASE_DATA[I] = VF_PRC_RobKor:BASE_DATA[I]
                ENDFOR
                ;zum testen nur Base4
                ;BASE_DATA[4] = VF_PRC_RobKor:BASE_DATA[4]
                  ;-------------Sensorkalibrierung-------------------
                N_PRC_MsgOff = 600
                N_PRC_Ret1   = PRC_MsgErr(#NotifyMsg,795)
                Repeat
                  B_PRC_ISTOOL = FALSE
                  N_PRC_Ret1   = PRC_MsgErr(#NotifyMsg,630)
                  REPEAT
                    N_PRC_Err1   = 0
                    B_PRC_MsgFlg = FALSE
                    N_PRC_Status = PRC_GetStatus()
                    PRC_DebugDlg(1,N_PRC_Status,0)
                    IF (N_PRC_Status <> 623) THEN ;kalibmode
                      N_PRC_Err1   = 632   ; Perceptron nicht in Kalibrier-Modus
                      B_PRC_MsgFlg = TRUE
                    ELSE
                      B_PRC_MsgFlg = FALSE
                      N_PRC_Ret1   = 1
                    ENDIF
                    IF B_PRC_MsgFlg THEN
                     N_PRC_Ret1 = PRC_MsgErr(#NotifyMsg,N_PRC_Err1)
                    ENDIF
                  UNTIL (N_PRC_Ret1 == 1)
                  IF (B_PRC_MsgFlg) THEN
                    $FLAG[F_PRC_Err] = TRUE
                    RETURN
                  ENDIF
                  N_PRC_ModNr = N_PRC_TmpCmpM
                  N_PRC_UpNr  = N_PRC_TmpCmpU
                  PRC_DebugDlg(26,0,0)
                  PRC_DebugDlg(25,N_PRC_ModNr,N_PRC_UpNr)
                  N_PRC_MsrErg = PRC_StartMsrPktMsr(N_PRC_ModNr,N_PRC_UpNr,nPAR6)
                  N_PRC_MsgOff = 600
                  IF B_PRC_MsgFlg THEN
                    N_PRC_Ret1       = PRC_MsgErr(#NotifyMsg,N_PRC_Err1)
                    $FLAG[F_PRC_Err] = TRUE
                    RETURN
                  ENDIF
                  SWITCH N_PRC_MsrErg
                    CASE 600,601  ;alles ok
                      ;N_PRC_Ret1 = PRC_MsgErr(#NotifyMsg,699)
                      $FLAG[F_PRC_NoErr] = TRUE
                      B_SensIsKalib = TRUE
                      B_PRC_TmpKalib = TRUE
                      N_PRC_RET1 = 2 ;damit wird nochmal pruefprogramm gefahren.
                    CASE 1152, 1156   ; Kalibrierung erforderlich
                      N_PRC_RET1 = 1
                    CASE 1153, 1154, 1157, 1158   ; Sensormontage pruefen
                      N_PRC_MsrErg = 610
                      N_PRC_Ret1   = PRC_MsgErr(#NotifyMsg,N_PRC_MsrErg)
                      IF N_PRC_Ret1 == 1 THEN
                        B_PRC_ISTOOL = FALSE
                        $FLAG[F_PRC_Err] = TRUE
                        RETURN
                      ENDIF
                    DEFAULT
                      N_PRC_Ret1 = PRC_MsgErr(#NotifyMsg,N_PRC_Err1)
                      B_PRC_ISTOOL = FALSE
                      $FLAG[F_PRC_Err] = TRUE
                      RETURN
                  ENDSWITCH
                Until B_SensIsKalib
                ;---------------ende Sensorkalibrierung-------------------
                N_PRC_MsgOff = 700
                N_PRC_RET1 = 0
              CASE 1151, 1154, 1155, 1158, 2000 ;Robotermontage pruefen
                N_PRC_MsrErg = 710
                N_PRC_Ret1 = PRC_MsgErr(#NotifyMsg,710)
                IF N_PRC_Ret1 == 1 THEN
                  B_PRC_ISBASE = FALSE
                  $FLAG[F_PRC_Err] = TRUE
                  RETURN
                ENDIF
              DEFAULT
                N_PRC_Ret1 = PRC_MsgErr(#NotifyMsg,N_PRC_Err1)
                B_PRC_ISBase = FALSE
                $FLAG[F_PRC_Err] = TRUE
                RETURN
            ENDSWITCH
          UNTIL (N_PRC_RET1 == 1)
          N_PRC_Ret1 = PRC_MsgErr(#NotifyMsg,798)
          $FLAG[F_PRC_NoErr] = TRUE
        CASE 1003 ;AutoGauge  ; Hauptgruppe 9, Untergruppe 3
          N_PRC_Ret1 = PRC_MsgErr(#NotifyMsg,910,FUNKTION,CMD_SEL)
        DEFAULT
          N_PRC_Ret1=PRC_MsgErr(#NotifyMsg,910,FUNKTION,CMD_SEL)
      ENDSWITCH
    CASE 551 ;Messen, Korrketurwerte abholen, Korrektur ausfuehren
      N_PRC_MsgOff = 1000
      B_PRC_MsgFlg = FALSE
      SWITCH CMD_SEL
        CASE 1002 ; RF  ; Hauptgruppe 9, Untergruppe 2
          REPEAT ;Wiederholen in T1 u. T2
            PRC_DebugDlg(6,0,0)
            PRC_DebugDlg(25,nPAR2,nPAR3)
            PRC_StartMessung(nPAR2,nPAR3,nPAR6)
            SWITCH N_PRC_Ret1
              CASE 1000
                ; OK
              CASE 1005,1006,1007,1008,1009,1011,1012,1043
                B_PRC_MsgFlg = TRUE
              DEFAULT
                B_PRC_MsgFlg = TRUE
            ENDSWITCH
            N_PRC_Ret1 = PRC_MsgErr(#NotifyMsg,N_PRC_Err1)
            IF N_PRC_Ret1 == 2 THEN
              N_PRC_MsgOff = 1000
              REPEAT
                PRC_DebugDlg(9,0,0)
                N_PRC_Err2 = PRC_Reset()
                N_PRC_Ret2 = PRC_MsgErr(#NotifyMsg,N_PRC_Err2)
              UNTIL (N_PRC_Ret2 == 1)
            ENDIF
          UNTIL (N_PRC_Ret1 == 1)
          IF (B_PRC_MsgFlg) THEN
            $FLAG[F_PRC_Err]   = TRUE
            RETURN
          ELSE
            $FLAG[F_PRC_NoErr] = TRUE
          ENDIF
          N_PRC_MsgOff = 1000
          PRC_DebugDlg(7,0,0)
          PRC_GetKorrektur(nPAR2,nPAR3,nPAR4,nPAR6)
          SWITCH N_PRC_Ret1
            CASE 1000
              ; OK
            CASE 1001,1017,1018,1027,1028,1038,1042,1043
              B_PRC_MsgFlg = TRUE
              RETURN
            DEFAULT
              B_PRC_MsgFlg = TRUE
          ENDSWITCH
          N_PRC_Ret1 = PRC_MsgErr(#NotifyMsg,N_PRC_Err1)
          N_PRC_MsgOff = 1000
          B_PRC_MsgFlg = FALSE
          SWITCH CMD_SEL
            CASE 1001,1002 ; IMT / RF  ; Hauptgruppe 9, Untergruppe 1 + 2
              ;wird im Advance erledigt
            CASE 1003 ;AutoGauge  ; Hauptgruppe 9, Untergruppe 3
              N_PRC_Ret1 = PRC_MsgErr(#NotifyMsg,910,FUNKTION,CMD_SEL)
            DEFAULT
              N_PRC_Ret1 = PRC_MsgErr(#NotifyMsg,910,FUNKTION,CMD_SEL)
          ENDSWITCH
        CASE 1003 ;AutoGauge  ; Hauptgruppe 9, Untergruppe 3
          N_PRC_Ret1 = PRC_MsgErr(#NotifyMsg,910,FUNKTION,CMD_SEL)
        DEFAULT
          N_PRC_Ret1 = PRC_MsgErr(#NotifyMsg,910,FUNKTION,CMD_SEL)
      ENDSWITCH
    CASE 552 ;Korrketurwerte abholen
      N_PRC_MsgOff = 1000
      B_PRC_MsgFlg = FALSE
      SWITCH CMD_SEL
        CASE 1002 ; RF  ; Hauptgruppe 9, Untergruppe 1 + 2
          PRC_DebugDlg(7,0,0)
          PRC_GetKorrektur(nPAR2,nPAR3,nPAR4,nPAR6)
          SWITCH N_PRC_Ret1
            CASE 1000
              ; OK
            CASE 1001,1017,1018,1027,1028,1038,1042,1043
              B_PRC_MsgFlg = TRUE
            DEFAULT
              B_PRC_MsgFlg = TRUE
          ENDSWITCH
          N_PRC_Ret1 = PRC_MsgErr(#NotifyMsg,N_PRC_Err1)
        CASE 1003 ;AutoGauge  ; Hauptgruppe 9, Untergruppe 3
          N_PRC_Ret1 = PRC_MsgErr(#NotifyMsg,910,FUNKTION,CMD_SEL)
        DEFAULT
          N_PRC_Ret1 = PRC_MsgErr(#NotifyMsg,910,FUNKTION,CMD_SEL)
      ENDSWITCH
    CASE 553 ;Korrketur ausfuehren
      N_PRC_MsgOff = 1000
      B_PRC_MsgFlg = FALSE
      SWITCH CMD_SEL
        CASE 1002 ; RF  ; Hauptgruppe 9, Untergruppe 1 + 2
          ;wird im Advance erledigt
        CASE 1003 ;AutoGauge  ; Hauptgruppe 9, Untergruppe 3
          N_PRC_Ret1 = PRC_MsgErr(#NotifyMsg,910,FUNKTION,CMD_SEL)
        DEFAULT
          N_PRC_Ret1 = PRC_MsgErr(#NotifyMsg,910,FUNKTION,CMD_SEL)
      ENDSWITCH
    CASE 554   ;korrektur holen + ausfuehren
      N_PRC_MsgOff = 1000
      B_PRC_MsgFlg = FALSE
      SWITCH CMD_SEL
        CASE 1002 ; RF  ; Hauptgruppe 9, Untergruppe 1 + 2
          PRC_DebugDlg(7,0,0)
          PRC_GetKorrektur(nPAR2,nPAR3,nPAR4,nPAR6)
          SWITCH N_PRC_Ret1
            CASE 1000
              ; OK
            CASE 1001,1017,1018,1027,1028,1038,1042,1043
              B_PRC_MsgFlg = TRUE
            DEFAULT
              B_PRC_MsgFlg = TRUE
          ENDSWITCH
          N_PRC_Ret1 = PRC_MsgErr(#NotifyMsg,N_PRC_Err1)
          N_PRC_MsgOff = 1000
          B_PRC_MsgFlg = FALSE
          PRC_DebugDlg(8,0,0)
          PRC_SetKorrektur(nPAR4)
          N_PRC_Ret1 = PRC_MsgErr(#NotifyMsg,N_PRC_Err1)
        CASE 1003 ;AutoGauge  ; Hauptgruppe 9, Untergruppe 3
          N_PRC_Ret1 = PRC_MsgErr(#NotifyMsg,910,FUNKTION,CMD_SEL)
        DEFAULT
          N_PRC_Ret1 = PRC_MsgErr(#NotifyMsg,910,FUNKTION,CMD_SEL)
      ENDSWITCH
    CASE 598 ;Perceptron reset
      SWITCH CMD_SEL
        CASE 1002,1003 ; RF / AG  ; Hauptgruppe 9, Untergruppe 1 + 2 + 3
          N_PRC_MsgOff = 500
          B_PRC_MsgFlg = FALSE
          PRC_DebugDlg(9,0,0)
          N_PRC_Err1   = PRC_Reset()
          N_PRC_Ret1   = 1
          N_PRC_Ret1   = PRC_MsgErr(#NotifyMsg,N_PRC_Err1)
          IF N_PRC_Err1 > 0 THEN
            $FLAG[F_PRC_Err]   = TRUE
          ELSE
            $FLAG[F_PRC_NoErr] = TRUE
          ENDIF
        DEFAULT
          N_PRC_Ret1 = PRC_MsgErr(#NotifyMsg,910,FUNKTION,CMD_SEL)
      ENDSWITCH
    CASE 599 ;Version
      SWITCH CMD_SEL
        CASE 1002,1003 ; RF / AG  ; Hauptgruppe 9, Untergruppe 1 + 2 + 3
          B_PRC_MsgKri = TRUE
          N_PRC_Ret1   = PRC_MsgErr(#NotifyMsg,9000)
        DEFAULT
          N_PRC_Ret1 = PRC_MsgErr(#NotifyMsg,910,FUNKTION,CMD_SEL)
      ENDSWITCH
  ENDSWITCH
END
;
  ;ENDFOLD (Main Programm)
;
  ;FOLD Start Punktmessung
;
DEFFCT INT PRC_StartMsrPktMsr(TYP:IN,SUBTYP:IN,PAR2:IN)
INT TYP
INT SUBTYP
INT PAR2
INT MsgOffset
BOOL bTypOk
  MsgOffset = N_PRC_MsgOff
  N_PRC_CurMod = TYP
  ; Modellkontrolle def. im Makro 57
  IF (TYP <= 0) OR (TYP == 10) OR (TYP == 20) OR ((TYP >= 30) AND (TYP <= 39)) OR (TYP > 42) THEN
    bTypOk       = FALSE
    N_PRC_Err1   = 872
    B_PRC_MsgFlg = TRUE
    B_PRC_MsgKri = TRUE
    N_PRC_Ret1   = PRC_MsgErr(#NotifyMsg,N_PRC_Err1,TYP)
    RETURN(N_PRC_Err1)
  ELSE
    bTypOk = BA_PRC_ModOn[TYP]
    IF bTypOk == FALSE THEN
       N_PRC_Err1   = 873
       B_PRC_MsgFlg = TRUE
       B_PRC_MsgKri = TRUE
       N_PRC_Ret1   = PRC_MsgErr(#NotifyMsg,N_PRC_Err1,TYP)
       RETURN(N_PRC_Err1)
    ENDIF
  ENDIF
  IF B_PRC_Ghost THEN
    N_PRC_Err1 = MsgOffset
    IF NA_PRC_UPNR[TYP,SUBTYP] > 0 THEN
      IF NA_PRC_UPNR[N_PRC_CurMod,N_PRC_UpNr] > 0 THEN
        SEL_RES = SELECT(#UP,NA_PRC_UPNR[N_PRC_CurMod,N_PRC_UpNr],TRUE)
        N_PRC_MsgOff = MsgOffset
        N_PRC_Err1   = MsgOffset
      ELSE
        N_PRC_Err1   = MsgOffset + 41
        B_PRC_MsgFlg = TRUE
        N_PRC_Ret1   = N_PRC_UpNr
        N_PRC_Ret1   = PRC_MsgErr(#NotifyMsg,N_PRC_Err1,N_PRC_CurMod,N_PRC_Ret1)
        RETURN(N_PRC_Err1)
      ENDIF
    ELSE
      N_PRC_Err1   = MsgOffset + 40
      B_PRC_MsgFlg = TRUE
      N_PRC_Ret1   = SUBTYP
      N_PRC_Ret1   = PRC_MsgErr(#NotifyMsg,N_PRC_Err1,TYP,N_PRC_Ret1)
    ENDIF
    RETURN(N_PRC_Err1)
  ENDIF
  REPEAT
    N_PRC_Err1   = MsgOffset
    B_PRC_MsgFlg = FALSE
    PRC_DebugDlg(6,0,0)
    PRC_DebugDlg(25,TYP,SUBTYP)
    PRC_StartMessung(TYP,SUBTYP,PAR2)
    IF N_PRC_Err1 <> MsgOffset THEN
      B_PRC_MsgFlg = TRUE
    ENDIF
    N_PRC_Ret1 = PRC_MsgErr(#NotifyMsg,N_PRC_Err1)
    IF N_PRC_Ret1 == 2 THEN
      REPEAT
        PRC_DebugDlg(9,0,0)
        N_PRC_Err2 = PRC_Reset()
        N_PRC_Ret2 = PRC_MsgErr(#NotifyMsg,N_PRC_Err2)
      UNTIL (N_PRC_Ret2 == 1)
    ENDIF
  UNTIL(N_PRC_Ret1 == 1)
  IF B_PRC_MsgFlg THEN
    RETURN(N_PRC_Err1)
  ENDIF
  N_PRC_CurMod = TYP
  N_PRC_UpNr   = N_PRC_P2Ack
  IF ((N_PRC_UpNr == 0) AND (NOT B_PRC_StrSPS)) THEN
    PRC_DebugDlg(4,0,0)
    PRC_MessungBeenden(1002)
    N_PRC_Ret1   = PRC_MsgErr(#NotifyMsg,N_PRC_Err1)
    N_PRC_Err1   = MsgOffset + 29   ; Routinennummer ist NULL
    B_PRC_MsgFlg = TRUE
    N_PRC_Ret1   = PRC_MsgErr(#NotifyMsg,N_PRC_Err1)
    RETURN(N_PRC_Err1)
  ENDIF
  WHILE N_PRC_UpNr <> 0
IF (NA_PRC_UPNR[TYP,SUBTYP] > 0) AND (bTypOk == TRUE) THEN
IF (NA_PRC_UPNR[N_PRC_CurMod,N_PRC_UpNr] > 0) AND (bTypOk == TRUE) THEN
        SEL_RES = SELECT(#UP,NA_PRC_UPNR[N_PRC_CurMod,N_PRC_UpNr],TRUE)
        B_PRC_MsgFlg = FALSE
        N_PRC_MsgOff = MsgOffset
        N_PRC_Err1   = MsgOffset
      ELSE
        N_PRC_Err1   = MsgOffset + 41
        B_PRC_MsgFlg = TRUE
        N_PRC_Ret1   = N_PRC_UpNr
        N_PRC_Ret1   = PRC_MsgErr(#NotifyMsg,N_PRC_Err1,N_PRC_CurMod,N_PRC_Ret1)
        IF (NOT B_PRC_StrSPS) THEN
          PRC_DebugDlg(4,0,0)
          ;korrekturen holen wenn Robotertausch
          if ((TYP == N_PRC_RobTaM) and (SUBTYP == N_PRC_RobTaU)) then
            PRC_GetKorrektur(TYP,SUBTYP,N_PRC_VFNr,PAR2)
          endif
          PRC_MessungBeenden(1002)
        ENDIF
        B_PRC_MsgFlg = TRUE
        RETURN(MsgOffset + 41)
      ENDIF
    ELSE
      N_PRC_Err1   = MsgOffset + 40
      B_PRC_MsgFlg = TRUE
      N_PRC_Ret1   = N_PRC_UpNr
      N_PRC_Ret1   = PRC_MsgErr(#NotifyMsg,N_PRC_Err1,N_PRC_CurMod,N_PRC_Ret1)
      IF (NOT B_PRC_StrSPS) THEN
        PRC_DebugDlg(4,0,0)
        ;korrekturen holen wenn Robotertausch
        if ((TYP == N_PRC_RobTaM) and (SUBTYP == N_PRC_RobTaU)) then
          PRC_GetKorrektur(TYP,SUBTYP,N_PRC_VFNr,PAR2)
        endif
        PRC_MessungBeenden(1002)
      ENDIF
      B_PRC_MsgFlg = TRUE
      RETURN(MsgOffset + 40)
    ENDIF
    IF (NOT B_PRC_StrSPS) THEN
      PRC_DebugDlg(4,0,0)
      ;korrekturen holen wenn Robotertausch
      if ((TYP == N_PRC_RobTaM) and (SUBTYP == N_PRC_RobTaU)) then
        PRC_GetKorrektur(TYP,SUBTYP,N_PRC_VFNr,PAR2)
        N_PRC_Err3 = N_PRC_Err1
      endif
      PRC_MessungBeenden(1001)
    ENDIF
    IF (((N_PRC_Err1 <> MsgOffset) AND (B_PRC_MsgFlg == TRUE)) OR ((N_PRC_UpNr == 0) AND (N_PRC_Err1 <> MsgOffset)) OR (N_PRC_Err3 <> 0)) THEN
      if (n_prc_err3 == 2000) then
         N_PRC_Err1 = N_PRC_Err3
      endif
      RETURN(N_PRC_Err1)
    ENDIF
  ENDWHILE
  RETURN(MsgOffset)
ENDFCT
;
  ;ENDFOLD (Start Punktmessung)
;
  ;FOLD Get Mess UP Nummer
;
DEFFCT INT PRC_GetMessUpNr(TYP:IN,SUBTYP:IN,PAR2:IN)
INT TYP
INT SUBTYP
INT PAR2
INT nAnzWdh
BOOL bTypOk
  N_PRC_Err1 = 800
  N_PRC_CurMod = TYP
  SUBTYP = 0
  ; Modellkontrolle def. im Makro 57
  IF (TYP <= 0) OR (TYP == 10) OR (TYP == 20) OR ((TYP >= 30) AND (TYP <= 39)) OR (TYP > 42) THEN
    bTypOk       = FALSE
    N_PRC_Err1   = 872
    B_PRC_MsgFlg = TRUE
    B_PRC_MsgKri = TRUE
    N_PRC_Ret1   = PRC_MsgErr(#NotifyMsg,N_PRC_Err1,TYP)
    RETURN(N_PRC_Err1)
  ELSE
    bTypOk = BA_PRC_ModOn[TYP]
    IF bTypOk == FALSE THEN
       N_PRC_Err1   = 873
       B_PRC_MsgFlg = TRUE
       B_PRC_MsgKri = TRUE
       N_PRC_Ret1   = PRC_MsgErr(#NotifyMsg,N_PRC_Err1,TYP)
       RETURN(N_PRC_Err1)
    ENDIF
  ENDIF
  IF B_PRC_Ghost THEN
    IF NA_PRC_UPNR[N_PRC_RobGhM,N_PRC_RobGhU] > 0 THEN
      IF NA_PRC_UPNR[N_PRC_CurMod,N_PRC_UpNr] > 0 THEN
        SEL_RES=SELECT(#UP,NA_PRC_UPNR[N_PRC_CurMod,N_PRC_UpNr],TRUE)
      ELSE
        N_PRC_Err1   = 841
        B_PRC_MsgFlg = TRUE
        N_PRC_Ret1   = N_PRC_UpNr
        B_PRC_MsgKri = TRUE
        N_PRC_Ret1   = PRC_MsgErr(#NotifyMsg,N_PRC_Err1,N_PRC_CurMod,N_PRC_Ret1)
        RETURN(N_PRC_Err1)
      ENDIF
    ELSE
      N_PRC_Err1   = 840
      B_PRC_MsgFlg = TRUE
      N_PRC_Ret1   = N_PRC_RobGhU
      B_PRC_MsgKri = TRUE
      N_PRC_Ret1   = PRC_MsgErr(#NotifyMsg,N_PRC_Err1,TYP,N_PRC_Ret1)
    ENDIF
    RETURN(N_PRC_Err1)
  ENDIF
  REPEAT
    nAnzWdh    = 0
    REPEAT
      nAnzWdh = nAnzWdh + 1
      PRC_StartUpMess(TYP,SUBTYP,PAR2)
      SWITCH N_PRC_Err1
        CASE 800
          ; OK
        CASE 801,805,806,807,808,809,811,817,818,827,828,843
          B_PRC_MsgFlg = TRUE
        DEFAULT
          B_PRC_MsgFlg = TRUE
      ENDSWITCH
      IF N_PRC_Err1 == 807 THEN
        wait sec 0.5
      ENDIF
    UNTIL ((N_PRC_Err1 <> 807) OR (nAnzWdh >= N_PRC_MaxAnz))
    IF nAnzWdh >= N_PRC_MaxAnz THEN
      B_PRC_MsgKri = TRUE
    ENDIF
    N_PRC_Ret1  = PRC_MsgErr(#NotifyMsg,N_PRC_Err1,N_PRC_CurMod,N_PRC_UpNr)
  UNTIL (N_PRC_Ret1 == 1)
  IF N_PRC_Err1 <> 800 THEN
    RETURN(N_PRC_Err1)
  ENDIF
  N_PRC_UpNr   = N_PRC_P2Ack
  N_PRC_CurMod = TYP
  IF (N_PRC_UpNr == 0) THEN
    N_PRC_Err1 = 829       ;Routinennummer ist NULL
    B_PRC_MsgKri = TRUE
    N_PRC_Ret1 = PRC_MsgErr(#NotifyMsg,N_PRC_Err1)
    RETURN(N_PRC_Err1)
  ENDIF
  IF NA_PRC_UPNR[N_PRC_CurMod,N_PRC_UpNr] > 0 THEN
    SEL_RES=SELECT(#UP,NA_PRC_UPNR[N_PRC_CurMod,N_PRC_UpNr],TRUE)
  ELSE
    N_PRC_Err1 = 841
    N_PRC_Ret1 = N_PRC_UpNr
    N_PRC_Ret1 = PRC_MsgErr(#NotifyMsg,N_PRC_Err1,N_PRC_CurMod,N_PRC_Ret1)
    B_PRC_MsgKri = TRUE
    RETURN(N_PRC_Err1)
  ENDIF
  RETURN(N_PRC_Err1)
ENDFCT
;
  ;ENDFOLD (Get Mess UP Nummer)
;
  ;FOLD Get Komp UP Nummer
;
DEFFCT INT PRC_GetKompUpNr(TYP:IN,SUBTYP:IN,PAR2:IN)
INT TYP
INT SUBTYP
INT PAR2
INT nAnzWdhErr        ; Anzahl der Wiederholungen im Fehlerfall (max 6, sh.dat)
INT nAnzWdhStat       ; Anzahl der Wiederholungen im Wartezustand (System noch im Messzyklus, aber Abbruch nach max. 60 + 2s)
BOOL bTypOk
  N_PRC_Err1   = 800
  N_PRC_CurMod = TYP
  ; Modellkontrolle def. im Makro 57
  IF (TYP <= 0) OR (TYP == 10) OR (TYP == 20) OR ((TYP >= 30) AND (TYP <= 39)) OR (TYP > 42) THEN
    bTypOk       = FALSE
    N_PRC_Err1   = 872
    B_PRC_MsgFlg = TRUE
    B_PRC_MsgKri = TRUE
    N_PRC_Ret1   = PRC_MsgErr(#NotifyMsg,N_PRC_Err1,TYP)
    RETURN(N_PRC_Err1)
  ELSE
    bTypOk = BA_PRC_ModOn[TYP]
    IF bTypOk == FALSE THEN
       N_PRC_Err1   = 873
       B_PRC_MsgFlg = TRUE
       B_PRC_MsgKri = TRUE
       N_PRC_Ret1   = PRC_MsgErr(#NotifyMsg,N_PRC_Err1,TYP)
       RETURN(N_PRC_Err1)
    ENDIF
  ENDIF
  IF B_PRC_Ghost THEN
    IF (NA_PRC_UPNR[N_PRC_RobGhM,N_PRC_RobGhU] > 0) AND (bTypOk == TRUE) THEN
      IF (NA_PRC_UPNR[N_PRC_CurMod,N_PRC_UpNr] > 0) AND (bTypOk == TRUE) THEN
        SEL_RES=SELECT(#UP,NA_PRC_UPNR[N_PRC_CurMod,N_PRC_UpNr],TRUE)
      ELSE
        N_PRC_Err1   = 841
        B_PRC_MsgFlg = TRUE
        N_PRC_Ret1   = N_PRC_UpNr
        B_PRC_MsgKri = TRUE
        N_PRC_Ret1   = PRC_MsgErr(#NotifyMsg,N_PRC_Err1,N_PRC_CurMod,N_PRC_Ret1)
        RETURN(N_PRC_Err1)
      ENDIF
    ELSE
      N_PRC_Err1   = 840
      B_PRC_MsgFlg = TRUE
      N_PRC_Ret1   = N_PRC_RobGhU
      B_PRC_MsgKri = TRUE
      N_PRC_Ret1   = PRC_MsgErr(#NotifyMsg,N_PRC_Err1,TYP,N_PRC_Ret1)
    ENDIF
    RETURN(N_PRC_Err1)
  ENDIF

  REPEAT
    nAnzWdhErr  = 0
    nAnzWdhStat = 0
    REPEAT
      PRC_StartUpKomp(TYP,SUBTYP,PAR2)

      SWITCH N_PRC_Err1
        CASE 800,850,851,852,853,860,861
          ; OK
        CASE 801,805,806,807,808,809,811,817,818,827,828,843,854,870,871
          B_PRC_MsgFlg = TRUE
        DEFAULT
          B_PRC_MsgFlg = TRUE
      ENDSWITCH

	  IF (N_PRC_Err1 == 860) OR (N_PRC_Err1 == 861) THEN
        wait sec 2
        nAnzWdhStat = nAnzWdhStat + 1
        IF nAnzWdhStat >= N_PRC_MaxSta THEN
          nAnzWdhErr = N_PRC_MaxErr
        ENDIF
      ELSE
        nAnzWdhErr = nAnzWdhErr + 1
      ENDIF
    UNTIL (((N_PRC_Err1 <> 860) AND (N_PRC_Err1 <> 861)) OR (nAnzWdhErr >= N_PRC_MaxErr))

	IF (nAnzWdhErr >= N_PRC_MaxErr) AND (B_PRC_Debug == TRUE) THEN
      B_PRC_MsgKri = TRUE
    ENDIF
    N_PRC_Ret1  = PRC_MsgErr(#NotifyMsg,N_PRC_Err1,N_PRC_CurMod,N_PRC_UpNr)
  UNTIL (N_PRC_Ret1 == 1)

  N_PRC_UpNr   = N_PRC_P2Ack

  IF (N_PRC_Err1 <> 851) AND (N_PRC_Err1 <> 852) THEN
    RETURN(N_PRC_Err1) ; keine Kompensation
  ENDIF

  IF (NA_PRC_UPNR[N_PRC_CurMod,N_PRC_UpNr] > 0) AND (bTypOk == TRUE) THEN
    SEL_RES=SELECT(#UP,NA_PRC_UPNR[N_PRC_CurMod,N_PRC_UpNr],TRUE)
  ELSE
    N_PRC_Err1 = 841
    N_PRC_Ret1 = N_PRC_UpNr
    N_PRC_Ret1 = PRC_MsgErr(#NotifyMsg,N_PRC_Err1,N_PRC_CurMod,N_PRC_Ret1)
    B_PRC_MsgKri = TRUE
    RETURN(N_PRC_Err1)
  ENDIF
  RETURN(N_PRC_Err1)
ENDFCT
;
  ;ENDFOLD (Get Komp UP Nummer)
;
  ;FOLD Get Status
;
DEFFCT INT PRC_GetStatus()
  N_PRC_ID     = 2

